# B&R Automation Studio project AS (part 2)

#### bgssm.c
```c
/********************************************************************
 * COPYRIGHT -- belgor
 ********************************************************************
 * Library: bglibas
 * File: bglibas.c
 * Author: admin
 * Created: March 07, 2012
 ********************************************************************
 * Implementation of library bglibas
 ********************************************************************/

#ifdef __cplusplus
  extern "C"
  {
#endif

#include <string.h>
// #include <stdarg.h>

#include  "bglibasWBR.h"                                                        //  WBR: could also keep the bglibas.h name and change the library's Properties->Library setting away from using the default name
#include  "bglibasWBR_C.h"

/* Init state machine. MUST be called once, before any other bgSSM function call. */
unsigned long bgSSMInit(struct bgSSM_typ* p, unsigned long pFunGetStateName, unsigned long pFunCyclicCallback)
{
  memset(p, 0, sizeof(struct bgSSM_typ));

  p->pfunGetStateName = (UDINT)pFunGetStateName;
  p->pfunCyclicCallback = (UDINT)pFunCyclicCallback;
  p->stateInit = 1;
  return(0);
}

/** Function pointer Init state machine. MUST be called once, before any other bgSSM function call. */
unsigned long bgSSMInitWbr(struct bgSSM_typ* p,                                    //  Pointer to state machine members and methods
                           unsigned long pfunInitState,                            //  Mandatory - initial method must be assigned
                           unsigned long pfunInterrupt,                            //  Optional
                           unsigned long pFunCyclicCallback)                       //  Optional
{
  memset(p, 0, sizeof(struct bgSSM_typ));

  p->pfunInitState=       (UDINT)pfunInitState;
  p->pfunInterrupt=       (UDINT)pfunInterrupt;
  p->pfunCyclicCallback=  (UDINT)pFunCyclicCallback;

  p->log.str.i.maxNodes=  200;
  p->log.str.list=  (linkedList_typ *)listSvcRequestList(BGSSM_MESSAGE_LENGTH_C,  lsQUEUE);

  p->stateNext= p->pfunInitState;                                                   //  WBR: assign init state function

  return(0);
}

/** State machine (SM) cyclic operation. */
unsigned long bgSSMCyclic(struct bgSSM_typ* p)
{
  int ii;

  //  TODO: implement interrupt/pause here to pause the delays with the SM

  //operate all timers
  for(ii=0; ii<BGSSM_TIMER_COUNT;ii++){
    bgTimerCyclic(&p->timer_x1ms[ii]);
  }
  bgTimerCyclic(&p->dlytimer_x1ms);
  bgTimerCyclic(&p->wdogTimer_x1ms);        //! \todo   log watchdog timeout \
                                                        provide automatic error state and go there? \
                                                        test func bgSSMStateNextWithWatchdog()

  //operate dlyCycle counter
  if(p->dlyCycles){
    p->dlyCycles--;
  }

  //call cyclic callback function if defined
  if(p->pfunCyclicCallback){
    void(*callback)(bgSSM_typ*) = ( void (*) (bgSSM_typ*) ) p->pfunCyclicCallback;
    (*callback)(p);
  }

  //clear single cycle flag every scan
  p->stateInit = 0;

  /// Evaluate breakpoint feature
  if(p->scanLimit.breakpoint && !p->scanLimit.active)   p->scanLimit.active=  1;          //  breakpoint has been found
  if(p->scanLimit.breakpointPrev && !p->scanLimit.breakpoint)   p->scanLimit.active=  0;  //  breakpoint switched off by

  /// Evaluate limit scan feature
  if(p->scanLimit.triggerNextScan)
  {
    p->scanLimit.triggerNextScan= p->scanLimit.count= 0;
  }
  if(!p->scanLimit.active)          memset(&p->scanLimit, 0, sizeof(p->scanLimit));
  else
  {
    if(p->scanLimit.count >= p->scanLimit.limit)   return 1;
    p->scanLimit.count++;
  }

  //check if state change requested
  if(p->state != p->stateNext){

    //if state change w. delay > wait for delay timer to expire or dlyCycles == 0
    if(!bgTimerIsTimeOut(&p->dlytimer_x1ms) || p->dlyCycles){                   //  TODO: add delay until event?
      return 1;
    }

    p->state = p->stateNext;
    //generate stateInit single scan flag
    p->stateInit = 1;

    //define state name if external function for state names is defined
    if( p->pfunGetStateName ){
      char*(*getStateName)(UDINT) = ( char* (*) (UDINT) )p->pfunGetStateName;
      strcpy(p->stateText, (*getStateName)(p->state));
    }else{
      strcpy(p->stateText, "???");
    }
  }

  if(p->pfunInitState)                                                          //  if the init state function pointer is defined...
  {
    void(*callState)(bgSSM_typ*) = ( void (*) (bgSSM_typ*) ) p->state;          //  ... call the function for the current state, i.e. use function pointer SM - WBR:
    (*callState)(p);
  }
  return(0);
}

/** SM state change methods
=============================*/

/** Change to next state. */
unsigned long bgSSMStateNext(struct bgSSM_typ* p, unsigned long stateNext)
{
  p->stateNext = stateNext;
  return(p->stateNext);
}

/** Store state to go to after SM subroutine. */
unsigned long bgSSMStateAfterSub(struct bgSSM_typ* p, unsigned long stateAfterSub)
{
  if(p->stateAfterSubIndex >= BGSSM_SUBROUTINE_COUNT)   return -99;     //  TODO: handle this error

  p->stateAfterSub[p->stateAfterSubIndex] = stateAfterSub;
  return(p->stateAfterSub[p->stateAfterSubIndex++]);
}

/** Activate state to go to after SM subroutine. */
unsigned long bgSSMReturnFromSub(struct bgSSM_typ* p)
{
  if(p->stateAfterSubIndex >= BGSSM_SUBROUTINE_COUNT)   return -99;     //  TODO: handle this error

  p->stateNext=    p->stateAfterSub[p->stateAfterSubIndex--];
  return(p->stateNext);
}

/** Change to next state w. timer delay. */
unsigned long bgSSMStateNextWithWatchdog(struct bgSSM_typ* p, unsigned long stateNext, unsigned long wdogTimeX1ms)
{
  p->stateNext = stateNext;
  bgTimerStart(&p->wdogTimer_x1ms, wdogTimeX1ms);
  return(p->stateNext);
}

/** Change to next state w. timer delay. */
unsigned long bgSSMStateNextTimeDelay(struct bgSSM_typ* p, unsigned long stateNext, unsigned long delayTimeX1ms)
{
  p->stateNext = stateNext;
  bgTimerStart(&p->dlytimer_x1ms, delayTimeX1ms);
  return(p->stateNext);
}

/** Change to next state w. cycles delay. */
unsigned long bgSSMStateNextCycleDelay(struct bgSSM_typ* p, unsigned long stateNext, unsigned long delayCycles)
{
  p->stateNext = stateNext;
  p->dlyCycles = delayCycles;
  return(p->stateNext);
}

/** Check if first scan for the state. */
plcbit bgSSMIsStateInit(struct bgSSM_typ* p)
{
  return(p->stateInit);
}

/** \todo  document */
UDINT  bgSSMPrintToTextLog(struct bgSSM_typ* p, const char* format, ...)
{
 va_list ap;

  va_start(ap, format);
  wbrvsnprintf((char *)listSvcRequestListNode(p->log.str.list), BGSSM_MESSAGE_LENGTH_C, format, ap);
  va_end(ap);

  return  listSvcCharListToStringArray(
                  p->log.str.list
                , &p->log.view[0][0]
                , BGSSM_MESSAGE_LENGTH_C
                , BGSSM_LOG_ENTRIES
                , p->log.str.i.offset
                , p->log.str.i.pageOffset
                , p->log.str.i.maxNodes
                , 1
                , ""
               );
}

/** \todo  document */
UDINT  bgSSMPrintLogMessage(struct bgSSM_typ* p)
{
  return  bgSSMPrintToTextLog(p, "%s", p->msg.log);
}

/** \todo  document */
UDINT  bgSSMPrintToTextLogIEC(struct bgSSM_typ* p, char* message)
{
  return  bgSSMPrintToTextLog(p, "%s", message);
}

/** \todo  document */
DINT  bgSSMPrintToLogbook(struct bgSSM_typ* p, const char* text, UDINT logIdent)
{
  return  requestMessageToLog( (UDINT)text, logIdent, 0, 0, 0, 0);              //  logIdent currently not used if logMsgType param is zero
}

/** \todo  document */
DINT  bgSSMPrintLogMessageToLogbook(struct bgSSM_typ* p, UDINT logIdent)    //! \todo   strcpy(loggermsg, requestedmsg) since msg gets destroyed, at least in ARsim
{
  return  requestMessageToLog( (UDINT)p->msg.log, logIdent, 0, 0, 0, 0);           //  logIdent currently not used if logMsgType param is zero
}

/** \todo  document */
DINT  bgSSMPrintToLogbookIEC(struct bgSSM_typ* p, char* message, UDINT logIdent)    //! \todo   strcpy(loggermsg, requestedmsg) since msg gets destroyed, at least in ARsim
{
  return  requestMessageToLog( (UDINT)message, logIdent, 0, 0, 0, 0);           //  logIdent currently not used if logMsgType param is zero
}

/** Check if first scan for the state.  If yes, perform some standard state change functions */
BOOL bgSSMIsStateInitWBR( struct bgSSM_typ* p                    //!  \todo   move this to C header
                        , /* const */ char* stateText            //!< This can take __FUNCTION__ or "text"
                        )
{
  if(p->stateInit)
  {
    if(stateText)  strcpy(p->stateText, stateText);
    wbrsnprintf(p->msg.log, sizeof(p->msg.log), "%s(%d)", bgSSMGetStateText(p), bgSSMGetState(p));      //! \todone? reserve p->message for other messages?
    bgSSMPrintToTextLog(p, "%s", p->msg.log);
    bgSSMPrintToLogbook(p, p->msg.log, 1);
  }

  return(p->stateInit);
}

/** SM data retrieval methods
=============================*/

/** Get current state */
unsigned long bgSSMGetState(struct bgSSM_typ* p)
{
  return(p->state);
}

/** Get current state text*/
plcstring* bgSSMGetStateText(struct bgSSM_typ* p)
{
  return(&p->stateText[0]);
}

#ifdef __cplusplus
  };
#endif
```

### Library Logical/UserLibraries/wbrServices/wbrPingSvc (ANSIC) - Ping a host or IP address
Depends on: AsICMP, wbrLogSvc, bglibasWBR, AsTime

### Package Logical/UserLibraries/wbrServices/wbrSvcUtilities - Utility functions

- Library Logical/UserLibraries/wbrServices/wbrSvcUtilities/wbrBitUtil (ANSIC) - Utilities for setting or extracting bits in bytes, words, ints, etc. (no source held here)

### wbrServicesGlobal.var - Global variables
```iecst
(********************************************************************
 * COPYRIGHT -- Piedmont Automation
 ********************************************************************
 * Package: listServices
 * File: listServicesGlobal.var
 * Author: Blanton Radford
 * Created: August 11, 2014
 ********************************************************************
 * Variables of package listServices
 ********************************************************************)
VAR
	memService : wbrMemService_typ := (0);
	logService : wbrLogService_typ := (0);
	genericPing : wbrPingService_typ;
	usbServiceIF : ARRAY[0..wbrusbLAST_NODE] OF wbrUSBServiceIF_typ;
END_VAR
```

### wbrServicesPackage.var - Package variables
```iecst
VAR
	usbService : wbrUSBService_typ;
END_VAR
```

### Package Logical/UserLibraries/wbrServices/InitSP - Place this program in TC#1 to initialize wbrServices

### paiConfig.typ
```iecst
(********************************************************************
 * COPYRIGHT --
 ********************************************************************
 * Package: ConfigAndRecipes
 * File: Config.typ
 * Author: goran_2
 * Created: August 06, 2011
 ********************************************************************
 * Data types of package ConfigAndRecipes
 ********************************************************************)
(*==================================================================*)
(*Config related structures that shall not be changed.*)
(*==================================================================*)

TYPE
	cfgConfig_enums :
		(
		ENUM_APPCFG_INFO_TEXT_LEN := 127,
		ENUM_APPCFG_PATHNAME_MAXLEN := 64,
		ENUM_APPCFG_PWD_MAXLEN := 15,
		ENUM_APPCFG_DEFECT_MAXINDEX := 11,
		ENUM_APPCFG_DEFECT_TXTMAXLEN := 31,
		ENUM_APPCFG_MAGIC_NUMBER := 16#55555555 (*Magic word (010101...) sequence (to detect battery backed up memory alterations)*)
		);
	cfgConfig_typ : 	STRUCT  (*Machine configuration includes settings for timers and settings for servo drives.*)
		cfgDefault : cfgMachineConfig_typ; (*The hardcoded defaults from the various application tasks.  This config should not be written to in the application code.  \todo  maintain a separate config that is the factory default config?*)
		machine : cfgMachineConfig_typ; (*The machine-level config.  Any item not set as product-level will use the value from this config.  When a different product is activated, this config will be copied to the active config first.*)
		recipe : cfgMachineConfig_typ; (*A holding space for a non-active recipe, i.e. product, config.  Possibly not needed or better located in the HMI package.  Would be used to support HMI editing of a product config that is not the active config.*)
		active : cfgMachineConfig_typ; (*The config used for current machine operation.  This will be the machine config*)
	END_STRUCT;
END_TYPE
```

### ConfigAndRecipes.var
```iecst
(********************************************************************
 * COPYRIGHT --
 ********************************************************************
 * Package: ConfigAndRecipes
 * File: ConfigAndRecipes.var
 * Author: goran_2
 * Created: August 06, 2011
 ********************************************************************
 * Variables of package ConfigAndRecipes
 ********************************************************************)
(*Constants*)
VAR CONSTANT
	APPCFG_DIRPATH_MAXLEN_IEC : DINT := 47;
	APPCFG_DIRPATH_MAXLEN_C : DINT := APPCFG_DIRPATH_MAXLEN_IEC + 1;
	APPCFG_FILENAME_MAXLEN_IEC : DINT := 63;
	APPCFG_FILENAME_MAXLEN_C : DINT := APPCFG_FILENAME_MAXLEN_IEC + 1;
	APPCFG_EXTENSION_MAXLEN_IEC : DINT := 15;
	APPCFG_EXTENSION_MAXLEN_C : DINT := APPCFG_EXTENSION_MAXLEN_IEC + 1;
	APPCFG_FULLPATH_MAXLEN_C : DINT := APPCFG_DIRPATH_MAXLEN_C + APPCFG_FILENAME_MAXLEN_C + APPCFG_EXTENSION_MAXLEN_C;
	APPCFG_FULLPATH_MAXLEN_IEC : DINT := APPCFG_FULLPATH_MAXLEN_C - 1;
END_VAR
(*Variables*)
VAR
	gConfig : cfgConfig_typ := (0); (*Machine configuration data*)
END_VAR
```

### Program Logical/UserLibraries/wbrServices/InitSP/runFirst (ANSIC) - Init wbrServices - PLACE IN TC#1 above most if not all other tasks

#### runFirstInit.c
```c
/*!
 ********************************************************************
 * Program : runFirst
 * \file :   runFirstInit.c
 * \author : Blanton Radford
 * \date Created: May 07, 2015
 * \copyright -- Piedmont Automation
 ********************************************************************
 * \brief Initializations for package WBRServices
 ********************************************************************/

#ifdef _DEFAULT_INCLUDES
  #include <AsDefault.h>
#endif

/*! \brief Init project compile info
*   called only from runFirstInit
*/
static void wbrServiceInitProgramCompileInfo()
{
 char osVers[12];
 TARGETInfo_typ TInfo;

  TInfo.enable = 1;
  TInfo.pOSVersion = (UDINT) &osVers;

  do {
    TARGETInfo(&TInfo);
  } while(TInfo.status == 0xFFFF);

#ifndef AS_PROJ
  #warning Macro names for program complile info not defined \
           -- code located just below this warning
  wbrsnprintf(gConfig.cfgDefault.cfgCompile.info, sizeof(gConfig.cfgDefault.cfgCompile.info), "No compile info");
  //* Copy the line below into Project->Change Runtime Versions->Build->ANSI C Build Options to define \
         -D "str(x)=#x" -D AS_PROJ=str($(AS_PROJECT_NAME)) -D AS_CFG=str($(AS_CONFIGURATION)) -D "AS_VERS=str($(AS_VERSION))" -D "AS_USER=str($(AS_USER_NAME))" -D "AS_CMPNY=str($(AS_COMPANY_NAME))" -D "AS_BUILD_MODE=str($(AS_BUILD_MODE))"

#else
  // These macro names are defined in Project->Change Runtime Versions->
  //    Build->ANSI C Build Options
  wbrsnprintf(gConfig.cfgDefault.cfgCompile.projVersion,  sizeof(gConfig.cfgDefault.cfgCompile.projVersion),  "%s, V1.0.00.6",  AS_PROJ);
  wbrsnprintf(gConfig.cfgDefault.cfgCompile.AS_config,    sizeof(gConfig.cfgDefault.cfgCompile.AS_config),    "%s",             AS_CFG);
  wbrsnprintf(gConfig.cfgDefault.cfgCompile.AS_configID,  sizeof(gConfig.cfgDefault.cfgCompile.AS_configID),  "%s_%s",          AS_PROJ, AS_CFG);
  wbrsnprintf(gConfig.cfgDefault.cfgCompile.AS_build,     sizeof(gConfig.cfgDefault.cfgCompile.AS_build),     "%s",             AS_BUILD_MODE);
  wbrsnprintf(gConfig.cfgDefault.cfgCompile.date,         sizeof(gConfig.cfgDefault.cfgCompile.date),         "%s @ %s",        __DATE__, __TIME__);
  wbrsnprintf(gConfig.cfgDefault.cfgCompile.AS_version,   sizeof(gConfig.cfgDefault.cfgCompile.AS_version),   "%s",             AS_VERS);
  wbrsnprintf(gConfig.cfgDefault.cfgCompile.user,         sizeof(gConfig.cfgDefault.cfgCompile.user),         "%s",             AS_USER);
  wbrsnprintf(gConfig.cfgDefault.cfgCompile.company,      sizeof(gConfig.cfgDefault.cfgCompile.company),      "%s, Inc.",       AS_CMPNY);
  wbrsnprintf(gConfig.cfgDefault.cfgCompile.info,         sizeof(gConfig.cfgDefault.cfgCompile.info),         "Compile info complete");
#endif
  wbrsnprintf(gConfig.cfgDefault.cfgCompile.AR_Version,   sizeof(gConfig.cfgDefault.cfgCompile.AR_Version),   "%s",           osVers);
  //! \todo   add WBRServices version, drawing name and revision, SVN revision
}

/*! \brief Init machine configuration defaults
*   called only from runFirstInit
*/
void  wbrMemServiceFirstInitSetDefaults(wbrMemSvcStoredConfig_typ* cfg)
{
  cfg->memRequestSize=   0xFFFFFF;

//  if(gREMMEMPostfix == 0x55555555)                                                 //  if storage has data, ...
//    cfg->memRequestSize=  (gRemanentData.activeCfg.wbrMemService.memRequestSize > 0xFFFFFF) ? gRemanentData.activeCfg.wbrMemService.memRequestSize : 0xFFFFFF;
  // if(magic == 0x55555555)                          //  if storage has data, ...
    // cfg->memRequestSize=  stored.wbrMemService.memRequestSize;
}

/*! \brief Init-SP for AsMem heap memory and linked list services
*   \pre   Place in TC#1 in front of most if not all other tasks
*/
void _INIT runFirstInit(void)
{
  wbrServiceInitProgramCompileInfo();

  //! \todo init AsMem as a separate service
  //! \todo what to do with appConfigAndRec - switch to MAPP?

  /// Init cfgDefault with hardcoded defaults
  if(&gConfig.cfgDefault.wbrMemService != 0)                   //  mcfgWBR: skip if this address is null    TODO: log this for debug
    memService.config= &gConfig.cfgDefault.wbrMemService;                //  mcfgWBR: this needs to run before the Config & Recipe task to insure the defaults are set

    // memService.config= &config.wbrMemService;                               //  mcfgWBR: used only for testing package independently

  wbrMemServiceFirstInitSetDefaults(memService.config);

  memService.status.memInitValid= initMemSvc(memService.config->memRequestSize);

  initListSvc(memService.status.memInitValid);

  setLogServiceDataAddress(&logService);

  if(memService.status.memInitValid)       initLogService();

  requestMessageToLogDefault( (UDINT)gConfig.cfgDefault.cfgCompile.projVersion);
  requestMessageToLogDefault( (UDINT)gConfig.cfgDefault.cfgCompile.AS_config);
  requestMessageToLogDefault( (UDINT)gConfig.cfgDefault.cfgCompile.AS_configID);
  requestMessageToLogDefault( (UDINT)gConfig.cfgDefault.cfgCompile.AS_build);
  requestMessageToLogDefault( (UDINT)gConfig.cfgDefault.cfgCompile.date);
  requestMessageToLogDefault( (UDINT)gConfig.cfgDefault.cfgCompile.AS_version);
  requestMessageToLogDefault( (UDINT)gConfig.cfgDefault.cfgCompile.AR_Version);
  requestMessageToLogDefault( (UDINT)gConfig.cfgDefault.cfgCompile.user);
  requestMessageToLogDefault( (UDINT)gConfig.cfgDefault.cfgCompile.company);
  requestMessageToLogDefault( (UDINT)gConfig.cfgDefault.cfgCompile.info);
  requestMessageToLogDefault( (UDINT)"wbrServices v0.12.0 initialized");
  requestSuccessEventToLog(
                        (UDINT)__FUNCTION__
                      , getSystemUserLogIdent()
                      , 0
                      , 50000
                      , 0
                      , (UDINT)"wbrServices v0.12.0 initialized"
                      , sizeof("wbrServices vn.nn.n initialized")
                      );

  wbrPingSvcInit(&genericPing);
}
```


### Package Logical/UserLibraries/wbrServices/TimerServices - ms-based time counters, pulses, etc.

### TimerServices.typ
```iecst
(********************************************************************
 * COPYRIGHT -- Piedmont Automation
 ********************************************************************
 * Package: TimerServices
 * File: TimerServices.typ
 * Author: Blanton Radford
 * Created: December 05, 2014
 ********************************************************************
 * Data types of package TimerServices
 ********************************************************************)

TYPE
	mstpPERIOD_enum :
		(
		per00100 := 0,
		per00200,
		per00500,
		per01000,
		per02000,
		per05000,
		per10000,
		perLAST
		);
	mstpFREQUENCY_enum :
		(
		freq010Hz := 0,
		freq005Hz,
		freq002Hz,
		freq001Hz,
		freq0p5Hz,
		freq0p2Hz,
		freq0p1Hz,
		freqLAST
		);
	mstpDUTY_CYCLE_enum :
		(
		duty01 := 0,
		duty10,
		duty20,
		duty25,
		duty50,
		dutyLAST
		);
	mstpDURATION_enum :
		(
		dur001ms := 0,
		dur010ms,
		dur020ms,
		durLAST
		);
	msTimerHourMeter_typ : 	STRUCT
		enable : BOOL;
		count : UDINT;
	END_STRUCT;
	msTmPulseSOS_typ : 	STRUCT
		codeSignal : BOOL;
		msgEnable : BOOL;
		shortEnable : BOOL;
		longEnable : BOOL;
		shortPulse : BOOL;
		longPulse : BOOL;
	END_STRUCT;
	msTmPulsePeriodDutyInOut_typ : 	STRUCT
		iPeriodValue : UDINT;
		iDutyValue : REAL;
		oPulse : BOOL;
	END_STRUCT;
	msTmPulseFreqDutyInOut_typ : 	STRUCT
		iFreqValue : REAL;
		iDutyValue : REAL;
		oPulse : BOOL;
	END_STRUCT;
	mstpPerDutyDurTableElements_typ : 	STRUCT
		duty : {REDUND_UNREPLICABLE} ARRAY[0..dutyLAST]OF BOOL;
		duration : {REDUND_UNREPLICABLE} ARRAY[0..durLAST]OF BOOL;
	END_STRUCT;
	msTimerPulse_typ : 	STRUCT
		periodDutyDurationTable : {REDUND_UNREPLICABLE} ARRAY[0..perLAST]OF mstpPerDutyDurTableElements_typ;
		periodLength : USINT;
		sos : msTmPulseSOS_typ;
	END_STRUCT;
	msTimer_typ : 	STRUCT
		pulse : msTimerPulse_typ; (*Various pulses calculated with ms precision (when allowed to by task class timing)*)
		initVal : UDINT; (*Initial value of clock_ms*)
		rolloverVal : UDINT;
		clock_ms : UDINT; (*System ms counter.  Not resettable.  Used to keep C1ms from missing counts if task class runs into its tolerance  TODO:  \todo*)
		diff_ms : UDINT; (*Difference from one scan to the next of the msTimeSvc task*)
		C1ms : UDINT; (*Rolls over after 4294920000U to keep other Cxx counters accurate.  Can also be reset.*)
		C10ms : UDINT;
		C100ms : UDINT;
		C1s : UDINT;
		C10s : UDINT;
		C60s : UDINT;
		C01sAbs : UDINT;
		C60sAbs : UDINT;
		F100ms : BOOL;
		F500ms : BOOL;
		F1s : BOOL;
		F2s : BOOL;
		F10s : BOOL;
		pulse01Hz100ms : BOOL;
		pulse1day100ms : BOOL;
		prev60s : UDINT;
		prev01s : UDINT;
	END_STRUCT;
END_TYPE
```

### Program Logical/UserLibraries/wbrServices/TimerServices/msTimeSvc (ANSIC)

#### msTimeSvc.c - Implementation code
```c
/*!
 ********************************************************************
### Program : msTimeSvc
 * \file :   msTimeSvc.c
 * \author : Blanton Radford
 * \date Created: December 05, 2014
 * \copyright -- Piedmont Automation
 ********************************************************************
 * \brief Implementation of program msTimeSvc
 ********************************************************************/

#ifdef _DEFAULT_INCLUDES
  #include <AsDefault.h>
#endif

_LOCAL BOOL running;    //  temporary
_LOCAL UDINT  run_ms;   //  temp

msTimer_typ * t=  &msTimer;

msTmPulsePeriodDutyInOut_typ  periodDutyDurationTable[perLAST][dutyLAST + durLAST]=
{
  {
      {  100,  1.0, 0}        //  period in ms, duty cycle in Hz, output
    , {  100, 10.0, 0}
    , {  100, 20.0, 0}
    , {  100, 25.0, 0}
    , {  100, 50.0, 0}
    , {  100, 01.0, 0}        //  period in ms, duty cycle in Hz, output
    , {  100, 10.0, 0}
    , {  100, 20.0, 0}
  }
 ,{
      {  200,  1.0, 0}        //  period, duty cycle, output
    , {  200, 10.0, 0}
    , {  200, 20.0, 0}
    , {  200, 25.0, 0}
    , {  200, 50.0, 0}
    , {  200, 01.0, 0}        //  period, duration, output
    , {  200, 10.0, 0}
    , {  200, 20.0, 0}
  }
 ,{
      {  500,  1.0, 0}        //  period, duty cycle, output
    , {  500, 10.0, 0}
    , {  500, 20.0, 0}
    , {  500, 25.0, 0}
    , {  500, 50.0, 0}
    , {  500, 01.0, 0}        //  period, duration, output
    , {  500, 10.0, 0}
    , {  500, 20.0, 0}
  }
 ,{
      { 1000,  1.0, 0}        //  period, duty cycle, output
    , { 1000, 10.0, 0}
    , { 1000, 20.0, 0}
    , { 1000, 25.0, 0}
    , { 1000, 50.0, 0}
    , { 1000, 01.0, 0}        //  period, duration, output
    , { 1000, 10.0, 0}
    , { 1000, 20.0, 0}
  }
 ,{
      { 2000,  1.0, 0}        //  period, duty cycle, output
    , { 2000, 10.0, 0}
    , { 2000, 20.0, 0}
    , { 2000, 25.0, 0}
    , { 2000, 50.0, 0}
    , { 2000, 01.0, 0}        //  period, duration, output
    , { 2000, 10.0, 0}
    , { 2000, 20.0, 0}
  }
 ,{
      { 5000,  1.0, 0}        //  period, duty cycle, output
    , { 5000, 10.0, 0}
    , { 5000, 20.0, 0}
    , { 5000, 25.0, 0}
    , { 5000, 50.0, 0}
    , { 5000, 01.0, 0}        //  period, duration, output
    , { 5000, 10.0, 0}
    , { 5000, 20.0, 0}
  }
 ,{
      {10000,  1.0, 0}        //  period, duty cycle, output
    , {10000, 10.0, 0}
    , {10000, 20.0, 0}
    , {10000, 25.0, 0}
    , {10000, 50.0, 0}
    , {10000, 01.0, 0}        //  period, duration, output
    , {10000, 10.0, 0}
    , {10000, 20.0, 0}
  }
}  ;

static  BOOL  pulsePeriodDurationWithOffset(
          UDINT per     //  period in ms
        , UDINT dur     //  Duration ( pulse on time) in ms
        , UDINT off     //  offset of start of pulse in ms
        )
{
  if(per < 2)   return  0;                                                      //  Period must be at least 2ms using ms precision
                                                                                //  Period must also be at least 2 * TC cycle time
  return  (   ((t->C1ms % per) >= off)
           && ((t->C1ms % per) < dur + off));
}

BOOL  getPulseOfPeriodAndDurationWithOffset(
          UDINT per     //  period in ms
        , UDINT dur     //  Duration ( pulse on time) in ms
        , UDINT off     //  offset of start of pulse in ms
        )
{
  return  pulsePeriodDurationWithOffset(per, dur, off);
}

BOOL  pulsePeriodDuration(
          UDINT per     //  period in ms
        , UDINT dur     //  Duration ( pulse on time) in ms
        )
{
  return  pulsePeriodDurationWithOffset(per, dur, 0);
}

BOOL  pulsePeriodDuty(
          UDINT per     //  period in ms
        , REAL  duty    //  duty cycle in %
        )
{
  if(duty <= 0.0)      return  0;                                                  //  Duty cycle must be greater than zero
  if(duty >= 100.0)    return  1;                                                  //  Signal always on if duty greater than 100%

  return  pulsePeriodDurationWithOffset(
                        per
                      , (UDINT)((REAL)per * duty / 100.0)
                      , 0
                      );
}

BOOL  pulseFreqDuty(
          REAL  f       //  frequency in Hz
        , REAL  d       //  duty cycle in %
        )
{
  if(d <= 0.0)      return  0;                                                  //  Duty cycle must be greater than zero
  if(f <= 0.0)      return  0;                                                  //  Prevent divide by zero
  if(f > 500.0)     return  0;                                                  //  Can't process higher frequencies using ms precision

  if(d >= 100.0)    return  1;                                                  //  Signal always on if duty greater than 100%

  return  pulsePeriodDurationWithOffset(
                        (UDINT)(1000.0 / f)
                      , ((UDINT)(1000.0 / f) * d / 100.0)
                      , 0
                      );
}

BOOL  pulseFreqDutyWithOffset(
          REAL  f       //  frequency in Hz
        , REAL  d       //  duty cycle in %
        , REAL  o       //  offset of start of pulse in %
        )
{
  if(d <= 0.0)      return  0;                                                  //  Duty cycle must be greater than zero
  if(f <= 0.0)      return  0;                                                  //  Prevent divide by zero
  if(f > 500.0)     return  0;                                                  //  Can't process higher frequencies using ms precision

  if(d >= 100.0)                  return  1;                                    //  Signal always on if duty greater than 100%
  if(o >= 100.0)                  return  0;                                    //  Signal always off if offset greater than 100%

  return  pulsePeriodDurationWithOffset(
                        (UDINT)(1000.0 / f)
                      , ((UDINT)(1000.0 / f) * d / 100.0)
                      , ((UDINT)(1000.0 / f) * o / 100.0)
                      );
}

BOOL  pulseFreqDuration(
          REAL  f       //  frequency in Hz
        , UDINT dur     //  Duration ( pulse on time) in ms
        )
{
  if((f <= 0.0) || (f > 500.0))   return  0;

  return  pulsePeriodDurationWithOffset(
                        (UDINT)(1000.0 / f)
                      , dur
                      , 0
                      );
}

BOOL  pulseFreqDurationWithOffset(
          REAL  f       //  frequency in Hz
        , UDINT dur     //  Duration ( pulse on time) in ms
        , UDINT off     //  offset of start of pulse in ms
        )
{
  if((f <= 0.0) || (f > 333.33))   return  0;

  return  pulsePeriodDurationWithOffset(
                        (UDINT)(1000.0 / f)
                      , dur
                      , off
                      );
}

/*! \brief Init-SP for millisecond timer services
*   \pre   Place in TC#1 or first used TC
*/
void _INIT msTimeSvcInit(void)
{

}

/*! \brief Cyclic task for millisecond timer services
*   \pre   Place in TC#1 or first used TC
*/
void _CYCLIC msTimeSvcCyclic(void)
{
 int  i, j;

  if(t->clock_ms == 0)    t->initVal= (UDINT)clock_ms();

  // if(<use external clock>)
  // t->clock_external=  <count from external source>;  i.e. a TC of < 1ms duration

  t->clock_ms=  (UDINT)clock_ms();

  t->diff_ms= t->clock_ms - t->C1ms - t->initVal;   //  Will this work at rollover?

  t->C1ms=  t->clock_ms - t->initVal; // + <rolloverVal>

  //! \todo   update C1ms in case task class runs into its tolerance \
              do this using a diff calc so that the function will continue to operate even if C1ms rolls over \
              OR just use clock_ms time and live with the rollover or implement a rollover counter

  /*! \todo
      if(<rolloverActive>)
        <rolloverVal>=  t->clock_ms - t->initVal + <prevRolloverVal> - 4294920000U;

      if( !<rolloverActive> && (t->C1ms > 4294920000U))
        <prevRolloverVal>=  <rolloverVal>;
        <rolloverVal>=  t->C1ms - 4294920000U;
        XX t->C1ms=  t->clock_ms=  0;      //  Keep absolute minute count accurate - WBR: check to see if this works
        XX -- OR --
        t->C1ms=  <rolloverVal>;      //  Keep absolute minute count accurate - WBR: check to see if this works
        t->C01sAbs++;
        t->C60sAbs++;
        rolloverActive= 1;

      //  This code will likely need to move ahead of t->diff_ms assignment
      if(t->clock_ms < t->C1ms)     //  rolled over
        t->initVal= (UDINT)clock_ms();
        <rolloverVal>+= t->diff_ms;  // assuming diff_ms works at rollover
        rolloverActive= 0;
        assign t->C1ms as above
  */
  // t->C1ms++;                                // inc ms counter
                                            // this will roll over after
                                            // 49.7102 days of continuous
                                            // running - WBR
                                            // resets with Start button

  /// Calculate Other Counters
  t->C10ms=   t->C1ms /   10;
  t->C100ms=  t->C1ms /  100;
  t->C1s=     t->C1ms / 1000;
  t->C10s=    t->C1ms / 10000;
  t->C60s=    t->C1ms / 60000;

  if(t->C1s  > t->prev01s)    t->C01sAbs++;       //  Rolls over after 136.193 years
  if(t->C60s > t->prev60s)    t->C60sAbs++;       //  Rolls over after 8171.55 years

  t->prev01s=  t->C1s;
  t->prev60s=  t->C60s;

  ///  Calc pulse trains
  //  <boolean>=    ((t->C1ms % <period>) < <duration>);      //  example - period and duration are in ms

  for(i=0; i<perLAST; i++)
  {
    for(j=0; j<dutyLAST; j++)
    {
      t->pulse.periodDutyDurationTable[i].duty[j]=
      periodDutyDurationTable[i][j].oPulse=
        pulsePeriodDuty(
            periodDutyDurationTable[i][j].iPeriodValue
          , periodDutyDurationTable[i][j].iDutyValue
          );
    }
    for( ; j < durLAST + dutyLAST; j++)
    {
      t->pulse.periodDutyDurationTable[i].duration[j - dutyLAST]=
      periodDutyDurationTable[i][j].oPulse=
        pulsePeriodDuration(
            periodDutyDurationTable[i][j].iPeriodValue
          , periodDutyDurationTable[i][j].iDutyValue
          );
    }
  }

  //  new
  t->pulse01Hz100ms= pulsePeriodDuration(1000, 100);                              //  add these in the application as needed, or put frequently used ones here
  t->pulse1day100ms= pulsePeriodDuration((24*3600*1000), 100);                    //  comes on once per day for 100ms

  t->pulse.sos.msgEnable=   pulseFreqDuty(0.25, 75.0);
  t->pulse.sos.shortEnable= pulseFreqDuty(0.50,  35.0);
  t->pulse.sos.longEnable=  pulseFreqDutyWithOffset(0.25, 17.5, 25.0);
  t->pulse.sos.shortPulse=  pulseFreqDuty( 4.0,  20.0);
  t->pulse.sos.longPulse=   pulseFreqDuty( 4.0,  60.0);

  t->pulse.sos.codeSignal=
    (   (t->pulse.sos.msgEnable && t->pulse.sos.shortEnable && t->pulse.sos.shortPulse)
     || (t->pulse.sos.msgEnable && t->pulse.sos.longEnable && t->pulse.sos.longPulse)) ;

  //  legacy
  t->F100ms=  pulsePeriodDurationWithOffset(  100,   50, 0);
  t->F500ms=  pulsePeriodDurationWithOffset(  500,  250, 0);
  t->F1s=     pulsePeriodDurationWithOffset( 1000,  500, 0);
  t->F2s=     pulsePeriodDurationWithOffset( 2000, 1000, 0);
  t->F10s=    pulsePeriodDurationWithOffset(10000, 5000, 0);

  //  TODO: add configurable, periodic pulse(s), i.e. an (n)s pulse every (nn)min or (nn)day(s) or ???
  //  TODO: add hour meter(s)
  if(running)
  {
    run_ms+=  t->diff_ms;
  }
}
```

### varPkg.var
```iecst
VAR
	gMachine : HERNON_Inline_Machine_typ;
	gMachineType : HERNON_Machine_Types_Enum;
END_VAR
```

### Disp_Global_Var.var
```iecst
VAR
	gHMITable_Rec_Dispense : hmiTableFBK_typ;
	gHMITable_Cfg_Dispense : hmiTableFBK_typ;
END_VAR
```

- Program Logical/Application_Logic/pkgDispense/Dispense (IEC) - Manage all dispense-valve related functionality (IO slice DS1) (no source held here)

### Library Logical/Application_Logic/pkgDispense/libDisp (IEC)

#### Disp_Rec_Cfg.typ
```iecst
TYPE
	HERNON_Rec_Dispense_typ : 	STRUCT
		Enable : UDINT;
		Disp_Valve_Edgemode_Pulse_TO_ms : REAL;
		Enable_Cure : UDINT;
		Extra_Shots_Per_VBlock : UDINT;
		Vblock_Offset_Additional_Shots : ARRAY[0..MAX_IDX_MULTIPLE_DISPENSE_SHOTS]OF REAL;
	END_STRUCT;
	HERNON_Cfg_Dispense_typ : 	STRUCT
		VBlock_Offset_From_PiP_Sensor : UDINT;
		Disp_Valve_Max_Output_High_TO_S : REAL;
		Disp_Signal_Reset_MaxTO_S : REAL;
		Disp_Valve_Max_RDY_NegEdge_S : REAL;
		Disp_Output_NegEdge_Margin_S : REAL;
	END_STRUCT;
END_TYPE
```

#### Disp_IO.typ
```iecst
TYPE
	X20DS4389_Edgegen_typ : 	STRUCT
		iEdgeMasterTime : DINT;
		iReadOutputStatus : BOOL;
		oEnableEdgeGen : BOOL;
		iEdgeGenReadbackEnabled : BOOL;
		oEdgeGenSequence : SINT;
		iEdgegenSequenceReadback : SINT;
		oEdgeGenTimestamp : DINT;
		iEdgeGenError : BOOL;
		oQuitEdgeGenError : BOOL;
		iEdgeGenWarning : BOOL;
		oQuitEdgeGenWarning : BOOL;
	END_STRUCT;
	HERNON_Inline_Dispense_Item_typ : 	STRUCT
		iValveReady : BOOL;
		oDispTrigger : BOOL;
		EdgeGen : X20DS4389_Edgegen_typ;
	END_STRUCT;
	HERNON_Inline_Dispense_IO_typ : 	STRUCT
		Projectile : HERNON_Inline_Dispense_Item_typ;
		Primer : HERNON_Inline_Dispense_Item_typ;
		iEdgeDetectError : BOOL;
		oQuitEdgeDetectError : BOOL;
	END_STRUCT;
END_TYPE
```

#### Disp_Alarms_Warnings.typ
```iecst
TYPE
	HERNON_Alarm_Dispense_typ : 	STRUCT
		Valve_Error_1 : BOOL; (*0*)
		Valve_Not_On : BOOL; (*1*)
		Valve_Not_OFF : BOOL; (*2*)
		Dispense_Reset_Error : BOOL; (*3*)
		Valve_Not_Off : BOOL; (*4*)
		Err_Disp_VBlock_Acc_Idx : BOOL; (*5*)
		Dispense_IO_Alloc_Error : BOOL; (*6*)
		Disp_Output_Not_Reset : BOOL; (*7*)
		Dispense_ValveRdy_NegEdge_Err : BOOL; (*8*)
		Disp_Valve_On_Too_Long : BOOL; (*9*)
		Dispense_Twice_Single_VBlock : BOOL; (*10*)
		ValveRdy_Not_Reset : BOOL; (*11*)
		Dispense_Not_Ready_On_Start : BOOL; (*12*)
		Dispense_Error_During_Runtime : BOOL; (*13*)
		VBlock_idx_during_shot_wait : BOOL; (*14*)
		VBlock_Offset_Invalid : BOOL; (*15*)
	END_STRUCT;
END_TYPE
```

### Insp_Global_Var.var
```iecst
VAR
	gHMITable_Rec_Inspect : hmiTableFBK_typ;
	gHMITable_Cfg_Inspect : hmiTableFBK_typ;
END_VAR
```

### Program Logical/Application_Logic/pkgInspect/Inspect (IEC)

#### Main.st - Init, cyclic, exit code
```iecst
//     __ __                         __  ___               ___         __           _             ____
//    / // /__ _______  ___  ___    /  |/  /__ ____  __ __/ _/__ _____/ /___ ______(_)__  ___ _  /  _/__  ____
//   / _  / -_) __/ _ \/ _ \/ _ \  / /|_/ / _ `/ _ \/ // / _/ _ `/ __/ __/ // / __/ / _ \/ _ `/ _/ // _ \/ __/
//  /_//_/\__/_/ /_//_/\___/_//_/ /_/  /_/\_,_/_//_/\_,_/_/ \_,_/\__/\__/\_,_/_/ /_/_//_/\_, / /___/_//_/\__(_)
//                                                                                      /___/
//  Copyright

PROGRAM _INIT
	Init_Logbook.Enable := TRUE;
	Init_Logbook.Name := 'usr_insp';
	Init_Logbook();

	gHMITable_Rec_Inspect(tableName := 'REC_INSPECT',		nameSpace := 'hmiTable/Rec/Inspect',	Logbook := Init_Logbook.pLog, 		pOverallStats := ADR(gTableStats.Overall));
	gHMITable_Cfg_Inspect(tableName := 'CFG_INSPECT',		nameSpace := 'hmiTable/Cfg/Inspect',	Logbook := Init_Logbook.pLog, 		pOverallStats := ADR(gTableStats.Overall));
END_PROGRAM

PROGRAM _CYCLIC

END_PROGRAM

PROGRAM _EXIT

END_PROGRAM
```

#### Variables.var - Local variables
```iecst
VAR
	FBK_Inspection_Camera : ARRAY[0..MAX_IDX_INSPECT_UNITS] OF Hernon_Inspection_Camera;
	Init_Logbook : FBK_Init_Logbook;
END_VAR
```

#### LocalFunctions.fun
```iecst
FUNCTION_BLOCK Hernon_Inspection_Camera (*TODO: Add your comment here*) (*$GROUP=User,$CAT=User,$GROUPICON=User.png,$CATICON=User.png*)
	VAR_INPUT
		pInspectionIO : REFERENCE TO HERNON_Inline_Inspect_Item_typ;
		pInspVBlock : REFERENCE TO VBlock_Object_typ;
		pInspRec : REFERENCE TO HERNON_Rec_Inspect_typ;
		pInspCfg : REFERENCE TO HERNON_Cfg_Inspect_typ;
		pInspStats : REFERENCE TO HERNON_Prcs_Stats_typ;
		pMechanics : REFERENCE TO HERNON_Cfg_Mechanics_typ;
		pInspSeqFails : REFERENCE TO UDINT;
		MachineState : Global_State_Enum;
		VBlock_Fractional_Position : REAL;
		Current_VBlock_At_PiP_Sensor : UDINT;
		idx_inspect_unit : USINT;
	END_VAR
	VAR
		InspVar_LastCycle : HERNON_Inspect_App_typ;
		InspVar : HERNON_Inspect_App_typ;
		Alarms : HERNON_Alarm_Inspect_typ;
	END_VAR
END_FUNCTION_BLOCK
```

#### FBK_Inspection_Camera.st
```iecst
(* TODO: Add your comment here *)
FUNCTION_BLOCK Hernon_Inspection_Camera

	InspVar.VBlock_At_Inspect_Unit := (Current_VBlock_At_PiP_Sensor + (pMechanics.N_VBlocks_Belt_Total - pInspCfg.VBlock_Offset_From_PiP_Sensor)) MOD (pMechanics.N_VBlocks_Belt_Total);
	InspVar.VBlock_Fract_Pos := VBlock_Fractional_Position;

	CASE InspVar.Status OF
		INSPECT_STATE_INIT:
			pInspectionIO.oInspectionTrigger := FALSE;
			pInspectionIO.oIlluminationTrigger := FALSE;

			InspVar.Status := INSPECT_STATE_READY;

		INSPECT_STATE_READY:
			IF pInspRec.Enable = 1 THEN //If inspection is enabled:
				IF (InspVar.VBlock_At_Inspect_Unit <> InspVar_LastCycle.VBlock_At_Inspect_Unit) THEN //Inspection VBlock index
					IF (pInspVBlock.VBlock_Is_Occupied AND pInspVBlock.Inspection[idx_inspect_unit].Item_Inspection_Status = INSPECTION_RESULTS_NONESOFAR) THEN //Current vblock in front of inspection after index is occupied and hasn't been inspected yet
						//Handle resetting the VC object array datapoints to restart recording
//						brsmemset(ADR(pInspVCTrend.iInspectionGood[0]), 0, MAX_IDX_DISPENSE_VC_ARRAY + 1);
//						brsmemset(ADR(pInspVCTrend.iInspectionBad[0]), 0, MAX_IDX_DISPENSE_VC_ARRAY + 1);
//						brsmemset(ADR(pInspVCTrend.iInspectionError[0]), 0, MAX_IDX_DISPENSE_VC_ARRAY + 1);
//						brsmemset(ADR(pInspVCTrend.oInspectionTrigger[0]), 0, MAX_IDX_DISPENSE_VC_ARRAY + 1);
//						brsmemset(ADR(pInspVCTrend.oIlluminationTrigger[0]), 0, MAX_IDX_DISPENSE_VC_ARRAY + 1);
						InspVar.ii_VC_Trend_idx := 0;

						InspVar.Status := INSPECT_STATE_WAIT_VBLOCK_DISP;

					ELSIF pInspVBlock.VBlock_Is_Occupied AND pInspVBlock.Inspection[idx_inspect_unit].Item_Inspection_Status <> INSPECTION_RESULTS_NONESOFAR THEN
//						pInspVBlock.Error.Inspection_Error_1 := TRUE;
						Alarms.Inspection_Error_1 := TRUE;
//						pInspVBlock.Inspection[ii_inspect_units].Item_Inspection_Status := INSPECTION_ERROR_ALREADY_DONE;
						InspVar.Status := INSPECT_STATE_ERROR;
					END_IF;
				ELSIF InspVar.Flag_Inspect_Trigger_Now THEN //Force inspection to occur, i.e. manual trigger
//					//Handle resetting the VC object array datapoints to restart recording
//					brsmemset(ADR(pInspVCTrend.iInspectionGood[0]), 0, MAX_IDX_DISPENSE_VC_ARRAY + 1);
//					brsmemset(ADR(pInspVCTrend.iInspectionBad[0]), 0, MAX_IDX_DISPENSE_VC_ARRAY + 1);
//					brsmemset(ADR(pInspVCTrend.iInspectionError[0]), 0, MAX_IDX_DISPENSE_VC_ARRAY + 1);
//					brsmemset(ADR(pInspVCTrend.oInspectionTrigger[0]), 0, MAX_IDX_DISPENSE_VC_ARRAY + 1);
//					brsmemset(ADR(pInspVCTrend.oIlluminationTrigger[0]), 0, MAX_IDX_DISPENSE_VC_ARRAY + 1);
					InspVar.ii_VC_Trend_idx := 0;

					InspVar.Flag_Inspect_Trigger_Now := FALSE;

					bgTimerStart(InspVar.Timer.Timer_Inspection_Illum_DO_High, Tms(pInspCfg.Insp_Illum_ON_TO_S));
					bgTimerStart(InspVar.Timer.Timer_Inspection_Trigger_Wait, Tms(pInspCfg.Insp_Trigger_Wait_TO_S));

					InspVar.Status := INSPECT_STATE_WAIT_TRIG; //When triggering insp. manually, skip straight to waiting for the triggers rather than waiting for the vblock fractional displacement.
				ELSIF pInspectionIO.iInspectionBusy THEN //Shouldn't get a busy signal when not expecting it
					Alarms.Inspection_Busy_Without_Signal := TRUE;
					InspVar.Status := INSPECT_STATE_ERROR;
				ELSIF NOT pInspectionIO.iInspectionRunning THEN //Should always see DI corresponding to "running" state
					Alarms.Inspection_Not_Running := TRUE;
					InspVar.Status := INSPECT_STATE_ERROR;
				END_IF;
			ELSE//Inspection is disabled:
				InspVar.Status := INSPECT_STATE_DISABLED;
			END_IF;

		INSPECT_STATE_WAIT_VBLOCK_DISP:
			pInspectionIO.oInspectionTrigger := FALSE;
			pInspectionIO.oIlluminationTrigger := FALSE;

			IF InspVar.VBlock_Fract_Pos > pInspRec.Insp_VBlock_Displacement  THEN
				bgTimerStart(InspVar.Timer.Timer_Inspection_Illum_DO_High, Tms(pInspCfg.Insp_Illum_ON_TO_S));
				bgTimerStart(InspVar.Timer.Timer_Inspection_Trigger_Wait, Tms(pInspCfg.Insp_Trigger_Wait_TO_S));
				InspVar.Status := INSPECT_STATE_WAIT_TRIG;
			END_IF;

		INSPECT_STATE_WAIT_TRIG:
			pInspectionIO.oInspectionTrigger := FALSE;
			pInspectionIO.oIlluminationTrigger := NOT bgTimerIsTimeOut(InspVar.Timer.Timer_Inspection_Illum_DO_High);

			IF bgTimerIsTimeOut(InspVar.Timer.Timer_Inspection_Trigger_Wait) THEN
				bgTimerStart(InspVar.Timer.Timer_Inspection_Trigger_DO_High, Tms(pInspRec.Insp_Trigger_ON_TO_S));
				bgTimerStart(InspVar.Timer.Timer_Max_Insp_Busy_Signal, Tms(pInspCfg.Inspection_Max_Busy_TO_S));
				//
				InspVar.Status := INSPECT_STATE_WAIT_BUSY;
			ELSIF InspVar.VBlock_At_Inspect_Unit <> InspVar_LastCycle.VBlock_At_Inspect_Unit THEN
				Alarms.Inspection_VBlock_Idx_Waiting := TRUE;
				InspVar.Status := INSPECT_STATE_ERROR;
			END_IF;

		INSPECT_STATE_WAIT_BUSY:
			pInspectionIO.oInspectionTrigger := NOT bgTimerIsTimeOut(InspVar.Timer.Timer_Inspection_Trigger_DO_High);
			pInspectionIO.oIlluminationTrigger := NOT bgTimerIsTimeOut(InspVar.Timer.Timer_Inspection_Illum_DO_High);

			IF pInspectionIO.iInspectionBusy THEN
				bgTimerStart(InspVar.Timer.Timer_Inspection_Results_Wait, Tms(pInspCfg.Insp_Results_Wait_TO_S));
				InspVar.Status := INSPECT_STATE_WAIT_RESULTS;
			ELSIF bgTimerIsTimeOut(InspVar.Timer.Timer_Max_Insp_Busy_Signal) THEN
				Alarms.Insp_Err_Max_Busy_TO := TRUE;
				InspVar.Status := INSPECT_STATE_ERROR;
			ELSIF InspVar.VBlock_At_Inspect_Unit <> InspVar_LastCycle.VBlock_At_Inspect_Unit THEN
				Alarms.Inspection_VBlock_Idx_Waiting := TRUE;
				InspVar.Status := INSPECT_STATE_ERROR;
			END_IF;

		INSPECT_STATE_WAIT_RESULTS:
			pInspectionIO.oInspectionTrigger := NOT bgTimerIsTimeOut(InspVar.Timer.Timer_Inspection_Trigger_DO_High);
			pInspectionIO.oIlluminationTrigger := NOT bgTimerIsTimeOut(InspVar.Timer.Timer_Inspection_Illum_DO_High);

			IF NOT pInspectionIO.iInspectionBusy THEN
				pInspectionIO.oInspectionTrigger := FALSE;
				pInspectionIO.oIlluminationTrigger := FALSE;
				IF pInspectionIO.iInspectionError AND NOT pInspectionIO.iInspectionGood THEN
					pInspVBlock.Inspection[idx_inspect_unit].Item_Inspection_Status := INSPECTION_RESULTS_ERROR;
					pInspStats.Num_Err := pInspStats.Num_Err + 1;
				ELSE
					IF pInspectionIO.iInspectionGood THEN
						pInspVBlock.Inspection[idx_inspect_unit].Item_Inspection_Status := INSPECTION_RESULTS_GOOD;
						pInspStats.Num_Passed := pInspStats.Num_Passed + 1;

						pInspSeqFails := 0;
					ELSE
						pInspVBlock.Inspection[idx_inspect_unit].Item_Inspection_Status := INSPECTION_RESULTS_BAD;
						pInspStats.Num_Failed := pInspStats.Num_Failed + 1;

						pInspSeqFails := pInspSeqFails + 1;
					END_IF;
				END_IF;
				pInspVBlock.Inspection[idx_inspect_unit].Inspection_Time := bgTimerTimeElapsed(InspVar.Timer.Timer_Inspection_Results_Wait);
				//Return to state to wait for next inspection trigger event
				InspVar.Status := INSPECT_STATE_READY;
			ELSIF bgTimerIsTimeOut(InspVar.Timer.Timer_Inspection_Results_Wait) THEN
				//Failed to receive results within the specified timeout
				pInspectionIO.oInspectionTrigger := FALSE;
				pInspectionIO.oIlluminationTrigger := FALSE;

				pInspStats.Num_Unanswered := pInspStats.Num_Unanswered + 1;

				Alarms.Inspection_Results_TO_NoAnswer := TRUE;
				InspVar.Status := INSPECT_STATE_ERROR;
			ELSIF InspVar.VBlock_At_Inspect_Unit <> InspVar_LastCycle.VBlock_At_Inspect_Unit THEN
				Alarms.Inspection_VBlock_Idx_Waiting := TRUE;
				InspVar.Status := INSPECT_STATE_ERROR;
			END_IF;

		INSPECT_STATE_ERROR:

		INSPECT_STATE_DISABLED:
			IF pInspRec.Enable = 1 THEN
				InspVar.Status := INSPECT_STATE_INIT;
			END_IF;
	END_CASE;

	//Call timers
	bgTimerCyclic(InspVar.Timer.Timer_Inspection_Trigger_DO_High);
	bgTimerCyclic(InspVar.Timer.Timer_Inspection_Illum_DO_High);
	bgTimerCyclic(InspVar.Timer.Timer_Inspection_Results_Wait);
	bgTimerCyclic(InspVar.Timer.Timer_Inspection_Trigger_Wait);
	bgTimerCyclic(InspVar.Timer.Timer_Max_Insp_Busy_Signal);
//	bgTimerCyclic(InspectionRunSigBypass_ResetTime);

END_FUNCTION_BLOCK
```

### Library Logical/Application_Logic/pkgInspect/libInsp (IEC)

#### Insp_Enumerations.typ
```iecst
TYPE
	HERNON_Inspect_Enum :
		(
		INSPECT_STATE_INIT := 0,
		INSPECT_STATE_READY := 1,
		INSPECT_STATE_WAIT_RESULTS := 2,
		INSPECT_STATE_ERROR := 3,
		INSPECT_STATE_DISABLED := 4,
		INSPECT_STATE_WAIT_TRIG := 5,
		INSPECT_STATE_WAIT_BUSY := 6,
		INSPECT_STATE_WAIT_VBLOCK_DISP := 7,
		INSPECT_STATE_MANUAL := 8
		);
	HERNON_Inspect_Unit_ID_Enum :
		(
		INSPECT_PRIMER := 0,
		INSPECT_MOUTH := 1
		);
	HERNON_Inspection_Outcome_Enum :
		(
		INSPECTION_RESULTS_NONESOFAR := 0,
		INSPECTION_RESULTS_GOOD := 1,
		INSPECTION_RESULTS_BAD := 2,
		INSPECTION_RESULTS_ERROR := 3,
		INSPECTION_NA_EMPTY_VBLOCK := 4,
		INSPECTION_ERROR_ALREADY_DONE := 5
		);
END_TYPE
```

#### Insp_RecCfg.typ
```iecst
TYPE
	HERNON_Rec_Inspect_typ : 	STRUCT
		Enable : UDINT;
		Insp_Trigger_ON_TO_S : REAL;
		Insp_VBlock_Displacement : REAL;
		Sequential_Fails_Stop_Line : UDINT;
	END_STRUCT;
	HERNON_Cfg_Inspect_typ : 	STRUCT
		VBlock_Offset_From_PiP_Sensor : UDINT;
		Inspection_Max_Busy_TO_S : REAL;
		Insp_Results_Wait_TO_S : REAL;
		Insp_Trigger_Wait_TO_S : REAL;
		Insp_Illum_ON_TO_S : REAL;
	END_STRUCT;
END_TYPE
```

#### Insp_Alarms_Warnings.typ
```iecst
TYPE
	HERNON_Alarm_Inspect_typ : 	STRUCT
		Inspection_Error_1 : BOOL; (*0,1*)
		Inspection_Error_2 : BOOL; (*2,3*)
		Inspect_IO_Alloc_Error : BOOL; (*4,5*)
		Err_Insp_VBlock_Acc_Idx : BOOL; (*6,7*)
		Inspection_Not_Running : BOOL; (*8,9*)
		Inspection_Busy_Without_Signal : BOOL; (*10,11*)
		Insp_Err_Max_Busy_TO : BOOL; (*12,13*)
		Inspection_Results_TO_NoAnswer : BOOL; (*14,15*)
		Inspection_VBlock_Idx_Waiting : BOOL; (*16,17*)
		Inspect_Not_Ready_On_Start : BOOL; (*18*)
		Inspect_Error_During_Runtime : BOOL; (*19*)
		Inspection_Sequential_Fails : BOOL; (*20,21*)
	END_STRUCT;
END_TYPE
```

### Program Logical/Application_Logic/Control

#### Main.st
```iecst
PROGRAM _INIT

END_PROGRAM

PROGRAM _CYCLIC
	(* Insert code here *)

	CASE MachineState OF
		MACHINE_STATE_INIT:

		MACHINE_STATE_IDLE:

		MACHINE_STATE_RUNNING:

		MACHINE_STATE_ERRORSTOP:

		MACHINE_STATE_MANUAL_CTRL:

	END_CASE;

	CASE ProcessState OF
		PRCS_STATE_INIT:

		PRCS_STATE_IDLE:

		PRCS_STATE_WAIT_LOADER:

		PRCS_STATE_FEED_OFFSET:

		PRCS_STATE_BLADE_CREASER:

		PROCESS_STATE_FINISHING:

		PROCESS_STATE_ERROR:

	END_CASE;
END_PROGRAM

PROGRAM _EXIT
	(* Insert code here *)

END_PROGRAM
```

### Program Logical/Application_Logic/FeedRoller

#### Main.st
```iecst
PROGRAM _INIT
	(* Insert code here *)

END_PROGRAM

PROGRAM _CYCLIC

END_PROGRAM

PROGRAM _EXIT
	(* Insert code here *)

END_PROGRAM
```

### Package Logical/paiComponents - pai Components and Libraries

### bgdebug.h
```c
#ifndef _BG_DEBUG_H
#define _BG_DEBUG_H

#ifdef WIN32
#define DBG printf
#define DBGMSG printf

#define DBGCRT printf
#define DBGERR printf
#define DBGWAR printf
#define DBGINF printf
#define DBGDBG printf

#else

#include <bur/plc.h>
#include "bgringbuffer.h"

#define BG_DEBUG_LEVEL_CRITICAL		0
#define BG_DEBUG_LEVEL_ERROR		1
#define BG_DEBUG_LEVEL_WARNING		2
#define BG_DEBUG_LEVEL_INFO			3
#define BG_DEBUG_LEVEL_DEBUG		4

#define BG_DEBUG_UNUSED	0x0

/*
- To completly remove debug msgs from the source code use:
#define BG_DEBUG_ENABLE 0
*/
#define BG_DEBUG_ENABLE 1

/*ptr to global ring buffer for debug messages*/
_GLOBAL bgRingBuffer_typ gRingBuffer;

#if BG_DEBUG_ENABLE == 1
/*BG_DEBUG_ENABLE == 1 => debug messages present in the source code*/
#define DBG(format, args...)	bgRingBuffPutDbgInfo(&gRingBuffer, __FILE__, __FUNCTION__, BG_DEBUG_LEVEL_CRITICAL, BG_DEBUG_UNUSED, format, ## args);
#define DBGMSG(format, args...)	bgRingBuffPrintf(&gRingBuffer, format, ## args);

#define DBGCRT(format, args...)	bgRingBuffPutDbgInfo(&gRingBuffer, __FILE__, __FUNCTION__, BG_DEBUG_LEVEL_CRITICAL, BG_DEBUG_UNUSED, format, ## args);
#define DBGERR(format, args...)	bgRingBuffPutDbgInfo(&gRingBuffer, __FILE__, __FUNCTION__, BG_DEBUG_LEVEL_ERROR, BG_DEBUG_UNUSED, format, ## args);
#define DBGWAR(format, args...)	bgRingBuffPutDbgInfo(&gRingBuffer, __FILE__, __FUNCTION__, BG_DEBUG_LEVEL_WARNING, BG_DEBUG_UNUSED, format, ## args);
#define DBGINF(format, args...)	bgRingBuffPutDbgInfo(&gRingBuffer, __FILE__, __FUNCTION__, BG_DEBUG_LEVEL_INFO, BG_DEBUG_UNUSED, format, ## args);
#define DBGDBG(format, args...)	bgRingBuffPutDbgInfo(&gRingBuffer, __FILE__, __FUNCTION__, BG_DEBUG_LEVEL_DEBUG, BG_DEBUG_UNUSED, format, ## args);

#else
/*BG_DEBUG_ENABLE == 0 => all debug messages removed from the source code*/
#define DBG(format, args...)  ;
#define DBGMSG(format, args...)  ;

#define DBGCRT(format, args...)	;
#define DBGERR(format, args...)	;
#define DBGWAR(format, args...)	;
#define DBGINF(format, args...)	;
#define DBGDBG(format, args...)	;

#endif /*#if BG_DEBUG_ENABLE*/

#endif /*#ifdef WIN32*/

#endif /*#ifndef _BG_DEBUG_H*/
```

### bgPVSerializeJSON.c
```c
#ifndef _BG_SERIALIZEJSON_C
#define _BG_SERIALIZEJSON_C
/**
3/17/2015
-fixed serious bug that was causing incorrect setting of the integer PV types shorter than DINT/UDINT (i.e. SINT, USINT, INT, UINT)
*/
#ifdef WIN32
#include "string.h"
#else
#include <bur/plctypes.h>
#endif

//#include <string.h>
//#include <brsystem.h>
//#include <sys_lib.h>
//#include <asstring.h>
#include "bgstring.h"
#include "bgsprintf.h"
#include "bgsscanf.h"
#include "bgsscanf.c"

#define PV_SERIALIZEJSON_ITEM_DELIM_CRLF "\r\n"
#define PV_SERIALIZEJSON_ITEM_DELIM_COMMA ","
//#define PV_SERIALIZE_STR_MARKUP "'"
#define PV_SERIALIZEJSON_STR_MARKUP "'"

#define PV_SERIALIZEJSON_ERR_ZEROPTR -1
#define PV_SERIALIZEJSON_ERR_PVNOTFOUND -2
#define PV_SERIALIZEJSON_ERR_PVADRNOTFOUND -3
#define PV_SERIALIZEJSON_ERR_OBUFOVERFLOW -4

#define PV_SERIALIZEJSON_ERR_LAST -10

typedef struct bgPVSerializeJSON_typ
{
	char* toOutStream;
	UDINT lengthOutStream;
	DINT outputCharCount;
	DINT errorCode;
	DINT arrayIndexFrom;
	DINT arrayIndexTo;
	char* pItemDelim;
	char* pStrMarkup;
	DINT lastElement;

}bgPVSerializeJSON_typ;

static void bgPVSubStructSerializeJSON(bgPVSerializeJSON_typ* p, char* pvNameRoot, char* pvName, UINT dimension);
static void bgPVSerializeJSON(bgPVSerializeJSON_typ* p, char* pvNameRoot, char* pvName);
static void bgPVArraySerializeJSONRootToFrom(bgPVSerializeJSON_typ* p, char* pvNameRoot, int dimension, int isArrayOfStruct);

//#ifndef DBG
//#define DBG() ;
//#endif

#define PV_TYPE_MAX_INDEX	24
static const char *bgPVTypeStrings[PV_TYPE_MAX_INDEX + 1]={
	"STRUCT",	/*0*/
	"BOOL",		/*1*/
	"SINT",		/*2*/
	"INT",		/*3*/
	"DINT",		/*4*/
	"USINT",		/*5*/
	"UINT",		/*6*/
	"UDINT",		/*7*/
	"REAL",		/*8*/
	"STRING ",	/*9*/
	"ULINT",		/*10*/
	"DATETIME",	/*11*/
	"TIME",		/*12*/
	"DATE",		/*13*/
	"LREAL",		/*14*/
	"ARRAY",		/*15*/
	"TIME_OF_DAY",	/*16*/
	"BYTE",		/*17*/
	"WORD",		/*18*/
	"DWORD",	/*19*/
	"LWORD",	/*20*/
	"WSTRING",	/*21*/
	"?22",		/*22*/
	"LINT",		/*23*/
	};

static const char *bgGetPVTypeString(int pvTypeIndex){
	if(pvTypeIndex >= PV_TYPE_MAX_INDEX){
		return "TYPE=?";
	}

	return bgPVTypeStrings[pvTypeIndex];
}

static void bgGetPVValueText(char* pvValue, UDINT data_typ, UDINT data_len, UINT dimension, UDINT adr)
{
/*
	if( dimension != 1)
		DBG("TODO: display multidimensional values...");
*/
	switch(data_typ){
		case PB_DT_STRUCT:
			//DBG("TODO: display struct values...");
			break;
		case PB_DT_BOOL:
			bgsprintf(pvValue, "%d", *( (char*)adr ));
			break;
		case PB_DT_INT8:
			bgsprintf(pvValue, "%d", *( (char*)adr) );
			break;
		case PB_DT_INT16:
			bgsprintf(pvValue, "%d", *( (short*)adr ) );
			break;
		case PB_DT_INT32:
			bgsprintf(pvValue, "%d", *( (int*)adr ));
			break;
		case PB_DT_BYTE:
			bgsprintf(pvValue, "%u", *( (unsigned char*)adr));
			break;
		case PB_DT_WORD:
			bgsprintf(pvValue, "%u", *( (unsigned short*)adr));
			break;
		case PB_DT_LONG:
			bgsprintf(pvValue, "%u", *( (unsigned int*)adr));
			break;
		case PB_DT_FLOAT:
			{
				char temp[32];
				ftoa( *((float*)adr), (UDINT)temp);
				bgsprintf(pvValue, "%s", temp);
			}
			break;
		case PB_DT_VIS:
			bgsprintf(pvValue, "%s", (char*)adr );
			break;
		case PB_DT_OCTET:
			//DBG("TODO: display octet values...");
			break;
		case PB_DT_DATE:
			//DBG("TODO: display date values...");
			break;
		case PB_DT_TIME:
			//DBG("TODO: display time values...");
			break;
		case PB_DT_DIFF:
			//DBG("TODO: display time-diff values...");
			break;
		case 14://double
			{
				char temp[32];
				double value_double = *((double*)(adr));
				float value_float = (float)value_double;
				ftoa( value_float, (UDINT)temp);
				bgsprintf(pvValue, "%s", temp);
			}
			break;
		case PB_DT_ARRAY:
			//DBG("TODO: display array values...");
			break;
	}
}

static void bgSetPVValueText(char* pvValue, UDINT data_typ, UDINT data_len, UINT dimension, UDINT adr)
{
/*
	if( dimension != 1)
		DBG("TODO: display multidimensional values...");
*/
	switch(data_typ){
		case PB_DT_STRUCT:
			//DBG("TODO: set struct values...");
			break;
		case PB_DT_BOOL:
			*((char*)adr) = (char)atoi((UDINT)pvValue);
			break;
		case PB_DT_INT8:
			*((SINT*)adr) = (SINT)atoi((UDINT)pvValue);
			break;
		case PB_DT_INT16:
			*((INT*)adr) = (INT)atoi((UDINT)pvValue);
			break;
		case PB_DT_INT32:
			*((DINT*)adr) = (DINT)atoi((UDINT)pvValue);
			break;
		case PB_DT_BYTE:
			*((USINT*)adr) = (USINT)atoi((UDINT)pvValue);
			break;
		case PB_DT_WORD:
			*((UINT*)adr) = (UINT)atoi((UDINT)pvValue);
			break;
		case PB_DT_LONG:
			*((UDINT*)adr) = (UDINT)atoi((UDINT)pvValue);
			break;
		case PB_DT_FLOAT:
			{
				*((float*)adr) = atof((UDINT)pvValue);
			}
			break;
		case PB_DT_VIS:
			{
				int ii=0;
				//copy string
				//don't copy over the size of the dest buffer!
				//terminate properly
				char* src=(char*)pvValue;
				char* dst=(char*)adr;
				//DBG("GBTST= %s len=%d", src, data_len);
				for(ii=0; ii<data_len; ii++){
					dst[ii] = src[ii];
					//if end of src string > exit
					if(!src[ii])
						break;
				}
				//src longer than dst > terminate dst
				dst[data_len-1] = 0;
			}
			break;
		case PB_DT_OCTET:
			//DBG("TODO: display octet values...");
			break;
		case PB_DT_DATE:
			//DBG("TODO: display date values...");
			break;
		case PB_DT_TIME:
			//DBG("TODO: display time values...");
			break;
		case PB_DT_DIFF:
			//DBG("TODO: display time-diff values...");
			break;
		case 14://double
			{
				float value_float = atof((UDINT)pvValue);
				double value_double = (double)value_float;
				*((double*)adr) = value_double;
			}
			break;
		case PB_DT_ARRAY:
			//DBG("TODO: display array values...");
			break;
	}
}

int bgFindCharInStrRev(char *s, char chr)
{
	int ii;
	int lenStr;
	char *ptrStr;

	/*exit if null ptrs*/
	if(!s)
		return -1;

	lenStr = strlen(s);

	/*exit if zero strings*/
	if( !lenStr || !chr )
		return -1;

	/*search for char <chr> within the string <s> starting from the end*/
	for(ii=lenStr-1; ii>=0; ii--)
	{
		ptrStr = s + ii;
		if(*ptrStr == chr){
			return (ii);
		}
	}
	return -1;
}

static void bgPVWriteOutStream(bgPVSerializeJSON_typ* p, char* pvName, char* pvTextValue)
{
	int dotPosition;

	if(!p || !p->toOutStream || !pvTextValue || !p->pItemDelim)
		return;

	if(pvName){
		dotPosition = bgFindCharInStrRev(pvName, '.');
		if(dotPosition < 0){
			dotPosition=0; //dot not found > take the entire pvname
		}else{
			dotPosition += 1;//dot found > take only the pvname after the dot
		}

		brsstrcat((UDINT)p->toOutStream, (UDINT)PV_SERIALIZEJSON_STR_MARKUP);
		brsstrcat((UDINT)p->toOutStream, (UDINT)&pvName[dotPosition]);
		brsstrcat((UDINT)p->toOutStream, (UDINT)PV_SERIALIZEJSON_STR_MARKUP);
		brsstrcat((UDINT)p->toOutStream, (UDINT)"=");
		brsstrcat((UDINT)p->toOutStream, (UDINT)pvTextValue);

		p->outputCharCount += brsstrlen((UDINT)pvName);
		p->outputCharCount += 1; //  + '='
	}else{
		brsstrcat((UDINT)p->toOutStream, (UDINT)pvTextValue);
	}

	if(!p->lastElement){
		brsstrcat((UDINT)p->toOutStream, (UDINT)p->pItemDelim);	// delimiter "\r\n" or ","
	}
	p->outputCharCount += strlen(pvTextValue);
	if(!p->lastElement){
		p->outputCharCount += strlen(p->pItemDelim); //  + sizeof the delimiter string
	}

	if(p->outputCharCount >= (p->lengthOutStream - 100) ){//TODO: needs to be a better way to handle output buffer overflow
		p->errorCode = PV_SERIALIZEJSON_ERR_OBUFOVERFLOW;
		return;
	}
}

static bgTxtWriteOutStream(bgPVSerializeJSON_typ* p, char* pTxt)
{
	if(!p || !p->toOutStream || !pTxt)
		return;

	brsstrcat((UDINT)p->toOutStream, (UDINT)pTxt);

	p->outputCharCount += strlen(pTxt);

	if(p->outputCharCount >= (p->lengthOutStream - 100) ){//TODO: needs to be a better way to handle output buffer overflow
		p->errorCode = PV_SERIALIZEJSON_ERR_OBUFOVERFLOW;
		return;
	}
}

static int bgPVSerializeJSONIsArray(int data_typ, int data_len, int dimension)
{
	if(data_typ && (dimension > 1)){
		return 1;
	}
	return 0;
}

static void bgPVArraySerializeJSON(bgPVSerializeJSON_typ* p, char* pvNameRoot, char* pvName, int dimension, int isArrOfStruct)
{
	char pvArrNameRoot[128];
	bgPVSerializeJSON_typ pvSerObj;

	if(!pvName)
		return;

	bgTxtWriteOutStream(p, PV_SERIALIZEJSON_STR_MARKUP);
	bgTxtWriteOutStream(p, pvName);
	bgTxtWriteOutStream(p, PV_SERIALIZEJSON_STR_MARKUP);
	bgTxtWriteOutStream(p, "=");

	pvSerObj.toOutStream = p->toOutStream;
	pvSerObj.lengthOutStream = p->lengthOutStream;
	pvSerObj.outputCharCount = p->outputCharCount;
	pvSerObj.errorCode = 0;
	pvSerObj.arrayIndexFrom = 0;
	pvSerObj.arrayIndexTo = dimension - 1;
	pvSerObj.pItemDelim =  PV_SERIALIZEJSON_ITEM_DELIM_COMMA;
	pvSerObj.pStrMarkup =  PV_SERIALIZEJSON_STR_MARKUP;
	pvSerObj.lastElement = 0;

	brsstrcpy((UDINT)pvArrNameRoot, (UDINT)pvNameRoot);
	brsstrcat((UDINT)pvArrNameRoot, (UDINT)".");
	brsstrcat((UDINT)pvArrNameRoot, (UDINT)pvName);

	bgPVArraySerializeJSONRootToFrom(&pvSerObj, pvArrNameRoot, dimension, isArrOfStruct);

	p->outputCharCount = pvSerObj.outputCharCount;
	p->errorCode = pvSerObj.errorCode;

}

static void bgPVArraySerializeJSONRootToFrom(bgPVSerializeJSON_typ* p, char* pvNameRoot, int dimension, int isArrayOfStruct)
{
	int ii = 0;
	// TODO: checking for max size of the strings that are copied to these arrays
	char structName[256];
	char structItemName[32];
	DINT arrLastElement;
/*
Array of objects:
 "myarray" = "[
 {ID=0, HeadID=0, var={Type=0, Format=0}},
 {},
 {}]"

*/

	arrLastElement = p->lastElement;
	p->lastElement = 0;
	bgTxtWriteOutStream(p, "[");
	for(ii = p->arrayIndexFrom; (ii < dimension) && (ii <= p->arrayIndexTo); ii++){
		// NOTE: verify why PV_item destroys content of the buffer supplied as 1st param
		{
			char arrayIndexTxt[10];
			brsstrcpy((UDINT)structItemName, (UDINT)pvNameRoot);
			brsstrcat((UDINT)structItemName, (UDINT)"[");
			brsitoa(ii, (UDINT)arrayIndexTxt);
			brsstrcat((UDINT)structItemName, (UDINT)arrayIndexTxt);
			brsstrcat((UDINT)structItemName, (UDINT)"]");
		}

		if(isArrayOfStruct)
			bgTxtWriteOutStream(p, "{");

		if((ii == (dimension-1)) || (ii == p->arrayIndexTo) ){
			p->lastElement = 1;
		}

		bgPVSerializeJSON(p, structItemName, 0);

		if((ii == (dimension-1)) || (ii == p->arrayIndexTo) ){
			if(isArrayOfStruct)
				bgTxtWriteOutStream(p, "}");
		}else{
			if(isArrayOfStruct)
				bgTxtWriteOutStream(p, "},");
		}

		if(p->errorCode)
			return;
	}

	if(!isArrayOfStruct){
		//	p->outputCharCount -= strlen(p->pItemDelim);//workaroud: remove delim for the last array element
		//	p->toOutStream[p->outputCharCount] = 0;
	}

	bgTxtWriteOutStream(p, "]");
	p->lastElement = arrLastElement;

	if(!isArrayOfStruct && !p->lastElement){
		bgTxtWriteOutStream(p, p->pItemDelim);
	}

}

static void bgPVSerializeJSON(bgPVSerializeJSON_typ* p, char* pvNameRoot, char* pvName)
{
	UINT status;
	UDINT data_typ;
	UDINT data_len;
	UINT dimension;
	UDINT adr;
	char structItemPVName[256];

	if( !pvName){
		brsstrcpy((UDINT)structItemPVName, (UDINT)pvNameRoot);

	}else{
		brsstrcpy((UDINT)structItemPVName, (UDINT)pvNameRoot);
		brsstrcat((UDINT)structItemPVName, (UDINT)".");
		brsstrcat((UDINT)structItemPVName, (UDINT)pvName);
	}

	status = PV_ninfo(structItemPVName, &data_typ, &data_len, &dimension);

	if( status ){
		p->errorCode = status;
		return;
	}

	if( bgPVSerializeJSONIsArray(data_typ, data_len, dimension) ){
		bgPVArraySerializeJSON(p, pvNameRoot, pvName, dimension, (data_typ==PB_DT_ARRAY)?1:0);
		return;
	}

	status = PV_xgetadr(structItemPVName, &adr, &data_len);

	if( status ){
		p->errorCode = status;
		return;
	}

	if( (data_typ == PB_DT_STRUCT) ){
		//DBG("PV='%s' Typ=%s Len=%d Dim=%d" , pvnamecomplete, bgGetPVTypeString(data_typ), data_len, dimension);

		if( (dimension == 1) && (data_len==4)){
			//enum data type!!! > will be handled below as a UDINT
			data_typ = PB_DT_INT32;
		}else{
			bgPVSubStructSerializeJSON(p, pvNameRoot, pvName, dimension);
			return;
		}
	}

	{
		char pvTextValue[256];
		int len = 0;

		if(data_typ == PB_DT_VIS){//STRING VALUES ONLY > marked with a special markup at the begining and end
			brsstrcpy((UDINT)pvTextValue, (UDINT)p->pStrMarkup);//set string begining markup (i.e. "\"")
			len = strlen(pvTextValue);
		}

		bgGetPVValueText(&pvTextValue[len], data_typ, data_len, dimension, adr);

		if(data_typ == PB_DT_VIS){//STRING VALUES ONLY > marked with a special markup at the begining and end
			brsstrcat((UDINT)pvTextValue, (UDINT)p->pStrMarkup);//set string ending markup (i.e. "\"")
		}

		//DBG("stritemPV='%s' Typ=%s Len=%d Dim=%d Val=%s" , pvName, bgGetPVTypeString(data_typ), data_len, dimension, pvTextValue);
		bgPVWriteOutStream(p, pvName, pvTextValue);
	}

}

static void bgPVSubStructSerializeJSON(bgPVSerializeJSON_typ* p, char* pvNameRoot, char* pvName, UINT dimension)
{
/*
Example:
typedef struct str1_typ{
UINT val1;
UINT val2;
}str1_typ;

typedef struct str2_typ{
UINT val3;
}str2_typ;

typedef struct str3_typ{
UINT val4;
struct str1_typ s1;
struct str2_typ s2;
}str3_typ;

_GLOBAL str3_typ test;

All available PV Names are:
test.val4
test.s1.val1
test.s1.val2
test.s2.val3;

Top PV Name (pvNameRoot):
test

During iteration, followin values will appear for 'structItemName':
s1
s2
val4

During iteration, following values will appear for 'structItemPVNameNoRoot':
val4
s1.val1
s1.val2
s2.val3

*/
	int ii = 0;
	// TODO: checking for max size of the strings that are copied to these arrays
	char structName[256];
	char structItemName[32];
	char structItemPVNameNoRoot[256];
	UINT status;
	UDINT data_typ;
	UDINT data_len;
	UDINT adr;

	if(pvName){
		bgTxtWriteOutStream(p, PV_SERIALIZEJSON_STR_MARKUP);
		bgTxtWriteOutStream(p, pvName);
		bgTxtWriteOutStream(p, PV_SERIALIZEJSON_STR_MARKUP);
		bgTxtWriteOutStream(p, "={");
	}

	for(ii=0; ii < dimension; ii++){
		// NOTE: verify why PV_item destroys concent of the buffer supplied as 1st param
		if( !pvName){
			brsstrcpy((UDINT)structName, (UDINT)pvNameRoot);
		}else{
			brsstrcpy((UDINT)structName, (UDINT)pvNameRoot);
			brsstrcat((UDINT)structName, (UDINT)".");
			brsstrcat((UDINT)structName, (UDINT)pvName);
		}

		//DBG("1)bgPVSubStr.. ii=%d str=%s item=%s", ii, structName, structItemName);
		status = PV_item(structName, ii, structItemName);
		//DBG("2)bgPVSubStr.. ii=%d str=%s item=%s", ii, structName, structItemName);

		if(status && (status != 14713)){
			// TODO: error handling
			//DBG("bgPVSubStr.. ii=%d str=%s item=%s err=%d", ii, structName, structItemName, status);
			p->errorCode = status;
			return;
		}

		//DBG("item=%d, name=%s", ii, structItemName);
		// TODO: check for max length of the PV name
		if(!pvName){
			brsstrcpy((UDINT)structItemPVNameNoRoot, (UDINT)structItemName);
		}else{
			if(status == 14713){//14713 is to handle enum type??? find out if there is a better solutiuon
				//following code is to handle an enum type that is reported as a structure (type 0). However, there are no structure elements and is not clear how to access values???
				char pvTextValue[64];

				status = PV_ninfo(structName, &data_typ, &data_len, &dimension);
				status = PV_xgetadr(structName, &adr, &data_len);
				//based on the reported lenght, try to guess the type of the enum
				if(data_len == 1){
					data_typ = PB_DT_BYTE;
				}else
					if(data_len == 2){
					data_typ = PB_DT_WORD;
				}else{
					data_typ = PB_DT_LONG;
				}
				bgGetPVValueText(&pvTextValue[0], data_typ, data_len, dimension, adr);
				if(ii == (dimension - 1)){
					p->lastElement = 1;
				}
				else{
					p->lastElement = 0;
				}
				bgPVWriteOutStream(p, pvName, pvTextValue);
				return;
			}

			brsstrcpy((UDINT)structItemPVNameNoRoot, (UDINT)pvName);
			brsstrcat((UDINT)structItemPVNameNoRoot, (UDINT)".");
			brsstrcat((UDINT)structItemPVNameNoRoot, (UDINT)structItemName);
		}

		if(ii == (dimension - 1)){
			p->lastElement = 1;
		}
		else{
			p->lastElement = 0;
		}
		bgPVSerializeJSON(p, pvNameRoot, structItemPVNameNoRoot);

		if(p->errorCode)
			return;
	}

	if(pvName){
		bgTxtWriteOutStream(p, "}");
	}
}

DINT bgPVRootArraySerializeJSON(char* pvNameRoot, char* toOutStream, UDINT lengthOutStream, UDINT begIndex, UDINT endIndex)
{
	UINT status;
	UDINT data_typ;
	UDINT data_len;
	UINT dimension;
	UDINT adr;
	DINT outputCharCount = 0;

	bgPVSerializeJSON_typ pvSerObj;

	if(!pvNameRoot || !toOutStream){
		return PV_SERIALIZEJSON_ERR_ZEROPTR;
	}

	if(toOutStream){
		brsstrcpy((UDINT)toOutStream, (UDINT)"");
	}
	pvSerObj.toOutStream = toOutStream;
	pvSerObj.lengthOutStream = lengthOutStream;
	pvSerObj.outputCharCount = 0;
	pvSerObj.errorCode = 0;
	pvSerObj.arrayIndexFrom = begIndex;
	pvSerObj.arrayIndexTo = endIndex;
	pvSerObj.pItemDelim =  PV_SERIALIZEJSON_ITEM_DELIM_COMMA;
	pvSerObj.pStrMarkup =  PV_SERIALIZEJSON_STR_MARKUP;
	pvSerObj.lastElement = 0;

	status = PV_ninfo(pvNameRoot, &data_typ, &data_len, &dimension);
	if( status ){
		return PV_SERIALIZEJSON_ERR_PVNOTFOUND;
	}

	status = PV_xgetadr(pvNameRoot, &adr, &data_len);
	if( status ){
		return PV_SERIALIZEJSON_ERR_PVADRNOTFOUND;
	}

	if(data_typ == PB_DT_STRUCT){
		//DBG("TOPPV='%s' Typ=%s Len=%d Dim=%d" , pvNameRoot, bgGetPVTypeString(data_typ), data_len, dimension);
		bgPVSubStructSerializeJSON(&pvSerObj, pvNameRoot, 0, dimension);
	}else
	if(data_typ == PB_DT_ARRAY){
		bgPVArraySerializeJSONRootToFrom(&pvSerObj, pvNameRoot, dimension, 1, 0);
	}else
	if(data_typ == PB_DT_VIS){//visible string
		bgPVArraySerializeJSONRootToFrom(&pvSerObj, pvNameRoot, dimension, 0, 1);
	}else
	if( ((data_typ == PB_DT_INT16) || (data_typ == PB_DT_INT32) || (data_typ == PB_DT_WORD) || (data_typ == PB_DT_LONG))&& (dimension > 1)){//aray of INT16
		bgPVArraySerializeJSONRootToFrom(&pvSerObj, pvNameRoot, dimension, 0, 1);
	}else{
		char pvTextValue[64];
		bgGetPVValueText(&pvTextValue[0], data_typ, data_len, dimension, adr);
		//DBG("TOPPV NOT A STRUCT! PV='%s' Typ=%s Len=%d Dim=%d Val=%s" , pvNameRoot, bgGetPVTypeString(data_typ), data_len, dimension, pvTextValue);
	}

	if(pvSerObj.errorCode){
		if(pvSerObj.errorCode < 0){
			return pvSerObj.errorCode;
		}
		return (pvSerObj.errorCode * (-1));
	}

	return pvSerObj.outputCharCount;
}

DINT bgPVStructSerializeJSON(char* pvNameRoot, char* toOutStream, UDINT lengthOutStream)
{
	UINT status;
	UDINT data_typ;
	UDINT data_len;
	UINT dimension;
	UDINT adr;
	DINT outputCharCount = 0;
	bgPVSerializeJSON_typ pvSerObj;

	if(!pvNameRoot || !toOutStream){
		return PV_SERIALIZEJSON_ERR_ZEROPTR;
	}

	if(toOutStream){
		brsstrcpy((UDINT)toOutStream, (UDINT)"");
	}
	pvSerObj.toOutStream = toOutStream;
	pvSerObj.lengthOutStream = lengthOutStream;
	pvSerObj.outputCharCount = 0;
	pvSerObj.errorCode = 0;
	pvSerObj.pItemDelim =  PV_SERIALIZEJSON_ITEM_DELIM_CRLF;
	pvSerObj.pStrMarkup =  "";

	status = PV_ninfo(pvNameRoot, &data_typ, &data_len, &dimension);
	if( status ){
		return PV_SERIALIZEJSON_ERR_PVNOTFOUND;
	}

	status = PV_xgetadr(pvNameRoot, &adr, &data_len);
	if( status ){
		return PV_SERIALIZEJSON_ERR_PVADRNOTFOUND;
	}

	if(data_typ == PB_DT_STRUCT){
		//DBG("TOPPV='%s' Typ=%s Len=%d Dim=%d" , pvNameRoot, bgGetPVTypeString(data_typ), data_len, dimension);
		bgPVSubStructSerializeJSON(&pvSerObj, pvNameRoot, 0, dimension);
	}else
	if(data_typ == PB_DT_ARRAY){
		pvSerObj.arrayIndexFrom = 0;
		pvSerObj.arrayIndexTo = dimension - 1;
		bgPVArraySerializeJSONRootToFrom(&pvSerObj, pvNameRoot, dimension, 1, 0);
	}
	else{
		char pvTextValue[64];
		bgGetPVValueText(&pvTextValue[0], data_typ, data_len, dimension, adr);
		//DBG("TOPPV NOT A STRUCT! PV='%s' Typ=%s Len=%d Dim=%d Val=%s" , pvNameRoot, bgGetPVTypeString(data_typ), data_len, dimension, pvTextValue);
	}

	if(pvSerObj.errorCode){
		if(pvSerObj.errorCode < 0){
			return pvSerObj.errorCode;
		}
		return (pvSerObj.errorCode * (-1));
	}

	return pvSerObj.outputCharCount;
}

//Maximum number of PV-s per file that can be deserialized!!!
#define BGPV_DESER_MAXPVCOUNT 1000

DINT bgPVStructDeserializeJSON(char* pvNameRoot, char* fromStream, UDINT lengthStream)
{
	UDINT ii;
	bgStringListEx_typ lineList1;
	bgStringListEx_typ lineSplit1;
	char* memLineList[BGPV_DESER_MAXPVCOUNT];
	char* memLineSplit[10];
	char structItemPVName[256];

	UINT status;
	UDINT data_typ;
	UDINT data_len;
	UINT dimension;
	UDINT adr;
	UDINT errorCounter = 0;

	bgStringListLinesEx(&lineList1, fromStream, (char*)memLineList, BGPV_DESER_MAXPVCOUNT*sizeof(char*));
	for(ii=0; ii<lineList1.itemCount; ii++){
		//DBG("ln%d: %s", ii, lineList1.items[ii]);
		bgStringSplitLineEx(&lineSplit1, '=',  (char*)lineList1.items[ii], (char*)memLineSplit, (int)10*sizeof(char*));
		//DBG("ln%d: key=%s val=%s", ii, lineSplit1.items[0], lineSplit1.items[1]);

		brsstrcpy((UDINT)structItemPVName, (UDINT)pvNameRoot);
		brsstrcat((UDINT)structItemPVName, (UDINT)".");
		brsstrcat((UDINT)structItemPVName, (UDINT)lineSplit1.items[0]);

		//DBG("PV=%s Val=%s", structItemPVName, lineSplit1.items[1]);
		status = PV_ninfo(structItemPVName, &data_typ, &data_len, &dimension);

		if( status ){
			// TODO: error handling
			//DBG("bgPVStructDes. PV='%s'; Error#=%d", structItemPVName, status);
			errorCounter++;
			continue;
		}

		status = PV_xgetadr(structItemPVName, &adr, &data_len);

		if( status ){
			// TODO: error handling
			//DBG("bgPVStructDes. Address for PV='%s'; Error=%d", structItemPVName, status);
			errorCounter++;
			continue;
		}

		bgSetPVValueText((char*)lineSplit1.items[1], data_typ, data_len, dimension, adr);
	}

	// TODO: return value in case of errors; detected version changes, etc.

	return errorCounter;

}

#endif //_BG_SERIALIZE_C
/*EOF*/
```

- Library Logical/paiComponents/Libraries/bgringbuf (ANSIC) (no source held here)

### Program Logical/paiComponents/paiFileService/paiFS (ANSIC) - pai File Service (TK#8)

#### paiFile.h - pai FS configuration defines 
```c
/********************************************************************
 * COPYRIGHT -- HP
 ********************************************************************
 * File: paiFile.h
 * Author: goran
 * Created: March 19, 2014
 *******************************************************************/

#include <bur/plctypes.h>

/*
###############################################################################
PAI_CONFIGURATION_SECTION
Code below allows configuration for:
application file system
###############################################################################
*/

/*
###############################################################################
Defines, Consts
###############################################################################
*/
/*
NOTE: Using C: disk is not the best solution considering that system files are there.
However, using disk other then C: (i.e. D:, etc) for application stuff creates
issue with the ability to view/copy/access application files from windows (multiple partitions not supported, etc)

File structure used in this application is following:

Directory:
C://Data
is used for application specific stuff.
This directory holds following files:
machine configuration file - "appcfg.txt"
machine factory deafult configuration file - "appcfgfactory.txt");

a subdirectory (REC) of the above directory is used for storing recipes.
C://Data/Rec

*/

#define PAI_FS_DEVICE_ROOT		"CFDISK"

/*file device name*/
//#define FILE_DEVICE_NAME	"CFDISK"
//#define FILE_DEVICE_CONF	 "/DEVICE=F:\\"
//#define FILE_DEVICE_CONF	 "/DEVICE=C:\\"
/*#define FILE_DEVICE_CONF	 "/DEVICE=D:\\Temp"*/

//IMPORTANT:
//in order for the following conditional compilation to work properly, PLC object in the Configuration view
//must contain following defintion:
//Folder: Build
//Field: Additional Build Options
//Value: -D $(AS_CONFIGURATION)
//Using the above, name of the current AS configuration (i.e. PPC820_ARwin1) becomes
//a defined preprocessor name. As a result, it's possible to destinguish between different configurations!
#ifdef PPC820_ARwin1
//In case of ARwin target, disk access uses networking and the disk storage is on the windows side
//CRITICAL NOTE: following IP address must match the Windows IP address within the ARWin networking configuration
//#define FILE_DEVICE_CONF "/SIP=192.168.1.15 /PROTOCOL=cifs /SHARE=abc /USER=abc /PASSWORD=abc"
#define FILE_DEVICE_CONF "/SIP=192.168.100.2 /PROTOCOL=cifs /SHARE=E_Data /USER=gainco /PASSWORD=gainco"
#warning "paiFS - ARwin target!"
#endif

#ifdef PPC820_ARwin
//In case of ARwin target, disk access uses networking and the disk storage is on the windows side
//CRITICAL NOTE: following IP address must match the Windows IP address within the ARWin networking configuration
//#define FILE_DEVICE_CONF "/SIP=192.168.1.15 /PROTOCOL=cifs /SHARE=abc /USER=abc /PASSWORD=abc"
#define FILE_DEVICE_CONF "/SIP=192.168.100.2 /PROTOCOL=cifs /SHARE=E_Data /USER=gainco /PASSWORD=gainco"
#warning "paiFS - ARwin target!"
#endif

//#ifndef FILE_DEVICE_CONF
#ifndef PAI_FS_DEVICE_ROOT_CFG
//For all other target (i.e ARsim and ARemb), storage resides on a physical disk present in the system
//#define FILE_DEVICE_CONF	 "/DEVICE=C:\\"
#define PAI_FS_DEVICE_ROOT_CFG	"/DEVICE=C:\\"
#warning "paiFS - NONE ARwin target!"
#warning "Please verify File System configuration in paiFS.h"
#endif

//===================================================================================
//Define application directories
//Dirs are located at PAI_FS_DEVICE_ROOT
#define PAI_FS_APP_DIR_DATA		"Data"
#define PAI_FS_APP_DIR_CFG		"Data/Cfg"
#define PAI_FS_APP_DIR_REC		"Data/Rec"

//===================================================================================
//Define application devices
//Devices are dedicated dirs at PAI_FS_DEVICE_ROOT to be used for specific purpose
#define PAI_FS_DEVICE_CFG	"CONFIG"
#define PAI_FS_DEVICE_CFG_CFG "/DEVICE=C:/Data/Cfg"

#define PAI_FS_DEVICE_REC	"RECIPES"
#define PAI_FS_DEVICE_REC_CFG "/DEVICE=C:/Data/Rec"

#define PAI_FS_DEVICE_REC_PALLETE	"FILESPALLETE"
#define PAI_FS_DEVICE_REC_PALLETE_CFG "/DEVICE=C:/Data/Rec/Pallets"

#define PAI_FS_DEVICE_REC_LAYER	"FILESLAYERS"
#define PAI_FS_DEVICE_REC_LAYER_CFG "/DEVICE=C:/Data/Rec/Layers"

#define PAI_FS_DEVICE_USB	"USB"
#define PAI_FS_DEVICE_USB_CFG "/DEVICE=C:/Data/Rec"
```

- Program Logical/paiComponents/paiFileService/paiFSUnitTest (ANSIC) - Example application code for using PAI file service. (no source held here)

### paiPVSerDesMgr.c - pai SerDes Manager
```c
/********************************************************************
 * COPYRIGHT --
 ********************************************************************
 * Package: paiFileService
 * File: paiPVSerDesMgr.c
 * Author: goran
 * Created: August 18, 2015
 *******************************************************************/

#include <bur/plctypes.h>
#ifdef _DEFAULT_INCLUDES
	#include <AsDefault.h>
#endif

#include "../bglib/bgPVSerialize.h"
#include "paiPVSerDesMgr.h"
#include "paiFSInterface.h"
/*
###############################################################################
Functions
###############################################################################
*/
/**
captureCurrentTimeStamp()
-captures current datetime, converts it to a string a places the result string into a user supplied
text buffer (pDst, dstSize)
*/
static void captureCurrentTimeStamp(char* pDst, UDINT dstSize)
{

	char txt_yyyy[8];
	char txt_mo[8];
	char txt_dd[8];
	char txt_hh[8];
	char txt_mm[8];
	char txt_ss[8];
	char txt_ms[8];

	if(!pDst)
		return;

	DTStructureGetTime_typ DTStrGetTime_1;
	DTStructure DTStruc;

	DTStrGetTime_1.enable = 1;
	DTStrGetTime_1.pDTStructure = (UDINT)&DTStruc;
	DTStructureGetTime(&DTStrGetTime_1);

	brsitoa(DTStruc.year, (UDINT)txt_yyyy);
	brsitoa(DTStruc.month, (UDINT)txt_mo);
	brsitoa(DTStruc.day, (UDINT)txt_dd);
	brsitoa(DTStruc.hour, (UDINT)txt_hh);
	brsitoa(DTStruc.minute, (UDINT)txt_mm);
	brsitoa(DTStruc.second, (UDINT)txt_ss);
	brsitoa(DTStruc.millisec, (UDINT)txt_ms);

	//sprintf(pDst, "%02d %02d %04d %02d:%02d:%02d", DTStruc.month, DTStruc.day, DTStruc.year, DTStruc.hour, DTStruc.minute, DTStruc.second);
	brsstrcpy((UDINT)pDst, (UDINT)txt_yyyy);
	brsstrcat((UDINT)pDst, (UDINT)"-");
	brsstrcat((UDINT)pDst, (UDINT)txt_mo);
	brsstrcat((UDINT)pDst, (UDINT)"-");
	brsstrcat((UDINT)pDst, (UDINT)txt_dd);
	brsstrcat((UDINT)pDst, (UDINT)" ");
	brsstrcat((UDINT)pDst, (UDINT)txt_hh);
	brsstrcat((UDINT)pDst, (UDINT)":");
	brsstrcat((UDINT)pDst, (UDINT)txt_mm);
	brsstrcat((UDINT)pDst, (UDINT)":");
	brsstrcat((UDINT)pDst, (UDINT)txt_ss);
	brsstrcat((UDINT)pDst, (UDINT)".");
	brsstrcat((UDINT)pDst, (UDINT)txt_ms);
}
/*
###############################################################################
PV Serialize / Deserialize Mgr
###############################################################################
*/

static void paiPVInitAtPowerUpCyclicSetStatus(char* pStatus, char* pText)
{
	brsstrcpy((UDINT)pStatus, (UDINT)pText);
}

static void paiPVInitAtPowerUpCyclic(paiPVSerDesMgr_typ* p)
{
	int ii;

	if(!p)
		return;

	for(ii=0; ii < p->iItemCount; ii++){
		if(p->pvItems[ii].optInitAtPowerUp.oInitReady)
			continue;

		//0-nothing to do
		if(p->pvItems[ii].optInitAtPowerUp.iPowerUpConfig == 0){
			p->pvItems[ii].optInitAtPowerUp.oInitReady = 1;
			paiPVInitAtPowerUpCyclicSetStatus(p->pvItems[ii].optInitAtPowerUp.oStatus, "off");
			continue;
		}

		//1-use test data, if diff, execute just default function
		if(p->pvItems[ii].optInitAtPowerUp.iPowerUpConfig == 1){
			//check test data validity
			if(!p->pvItems[ii].optInitAtPowerUp.pTestDataStorage ||
				!p->pvItems[ii].optInitAtPowerUp.iTestData){
				p->pvItems[ii].optInitAtPowerUp.oError = 1;
				continue;
			}

			//check if callback function defined
			if(!p->pvItems[ii].pCallbackDefault){
				p->pvItems[ii].optInitAtPowerUp.oError = 2;
				continue;
			}

			//compare test data
			if( (*(UDINT*)(p->pvItems[ii].optInitAtPowerUp.pTestDataStorage)) != p->pvItems[ii].optInitAtPowerUp.iTestData ){
				//difference!!! > execute default function
				void (*fDefault)() =  ( void(*) () ) p->pvItems[ii].pCallbackDefault;
				(*fDefault)();
				p->pvItems[ii].optInitAtPowerUp.oInitReady = 1;
				paiPVInitAtPowerUpCyclicSetStatus(p->pvItems[ii].optInitAtPowerUp.oStatus, "test+dflt");
			}else{
				p->pvItems[ii].optInitAtPowerUp.oInitReady = 1;
				paiPVInitAtPowerUpCyclicSetStatus(p->pvItems[ii].optInitAtPowerUp.oStatus, "test+n.a.");
			}

			//write test data to data storage
			*((UDINT*)p->pvItems[ii].optInitAtPowerUp.pTestDataStorage) = p->pvItems[ii].optInitAtPowerUp.iTestData;
			continue;
		}

		//2-use test data, if diff, execute default function then restore data from file
		if(p->pvItems[ii].optInitAtPowerUp.iPowerUpConfig == 2){
			//check test data validity
			if(!p->pvItems[ii].optInitAtPowerUp.pTestDataStorage ||
			!p->pvItems[ii].optInitAtPowerUp.iTestData){
				p->pvItems[ii].optInitAtPowerUp.oError = 1;
				continue;
			}

			//check if callback function defined
			if(!p->pvItems[ii].pCallbackDefault){
				p->pvItems[ii].optInitAtPowerUp.oError = 2;
				continue;
			}

			//compare test data
			if( *((UDINT*)p->pvItems[ii].optInitAtPowerUp.pTestDataStorage) != p->pvItems[ii].optInitAtPowerUp.iTestData ){
				//difference!!! > execute default function
				void (*fDefault)() =  ( void(*) () ) p->pvItems[ii].pCallbackDefault;
				(*fDefault)();
				//p->pvItems[ii].optInitAtPowerUp.oInitReady = 1;
				paiPVInitAtPowerUpCyclicSetStatus(p->pvItems[ii].optInitAtPowerUp.oStatus, "test+dflt");
				//now, request read from file
				p->pvItems[ii].iDesRequest = 1;
			}else{
				paiPVInitAtPowerUpCyclicSetStatus(p->pvItems[ii].optInitAtPowerUp.oStatus, "test+n.a.");
				p->pvItems[ii].optInitAtPowerUp.oInitReady = 1;
			}

			//write test data to data storage
			*((UDINT*)p->pvItems[ii].optInitAtPowerUp.pTestDataStorage) = p->pvItems[ii].optInitAtPowerUp.iTestData;
			continue;
		}
	}
}

static void paiPVChangeMonitorInit(paiPVSerDesMgr_typ* p)
{

}

static void paiPVChangeMonitorCyclic(paiPVSerDesMgr_typ* p)
{
int ii;

	if(!p)
		return;

	for(ii=0; ii < p->iItemCount; ii++){

		//HMI DesRequest (i.e. Read PV from file request via HMI)
		if(!p->pvItems[ii].iDesRequest && (p->pvItems[ii].optPtrHMIData && p->pvItems[ii].optPtrHMIData->iBtnDesRequest)){
			p->pvItems[ii].optPtrHMIData->iBtnDesRequest = 0;
			p->pvItems[ii].iDesRequest = 1;
			continue;
		}

		//HMI SerRequest (i.e. Write PV to file request via HMI)
		if(!p->pvItems[ii].iSerRequest && (p->pvItems[ii].optPtrHMIData && p->pvItems[ii].optPtrHMIData->iBtnSerRequest)){
			p->pvItems[ii].optPtrHMIData->iBtnSerRequest = 0;
			p->pvItems[ii].iSerRequest = 1;
			continue;
		}

		//check if feature PV change monitoring feature is enabled for an item
		if(!p->pvItems[ii].optChangeMonitor.iChngEnable)
			continue;

		if(!p->pvItems[ii].pPV || !p->pvItems[ii].iPVSize){
			p->pvItems[ii].optChangeMonitor.oError = 3;
			continue;
		}

		if(!p->pvItems[ii].optChangeMonitor.pChangeMonitorMem){
			p->pvItems[ii].optChangeMonitor.oError = 1;
			continue;
		}

		if(p->pvItems[ii].iPVSize > p->pvItems[ii].optChangeMonitor.iChangeMonitorMemSize ){
			p->pvItems[ii].optChangeMonitor.oError = 2;
			continue;
		}

		if(p->pvItems[ii].optChangeMonitor.oState == 0){
			//init state > copy PV to private memory, begin change monitor
			brsmemcpy((UDINT)p->pvItems[ii].optChangeMonitor.pChangeMonitorMem, (UDINT)p->pvItems[ii].pPV, p->pvItems[ii].iPVSize);

			p->pvItems[ii].optChangeMonitor.iChngAccepted = 0;
			p->pvItems[ii].optChangeMonitor.iChngRejected = 0;
			p->pvItems[ii].optChangeMonitor.oChngDetected = 0;

			p->pvItems[ii].optChangeMonitor.oState = 1;
		}

		if(p->pvItems[ii].optChangeMonitor.oState == 1){

			//working state > monitor PV changes
			if( !brsmemcmp((UDINT)p->pvItems[ii].optChangeMonitor.pChangeMonitorMem, (UDINT)p->pvItems[ii].pPV, p->pvItems[ii].iPVSize) ){
				p->pvItems[ii].optChangeMonitor.oChngDetected = 0;
				if(p->pvItems[ii].optPtrHMIData){
					//HMI is defined
					p->pvItems[ii].optPtrHMIData->oBtnVisible = 1;//not visible
				}
				continue;
			}
			//change detected!
			p->pvItems[ii].optChangeMonitor.oChngDetected = 1;
			if(p->pvItems[ii].optPtrHMIData){
				//HMI is defined
				p->pvItems[ii].optPtrHMIData->oBtnVisible = p->pvItems[ii].optChangeMonitor.oChngDetected ? 0 : 1;
			}

			if(p->pvItems[ii].optChangeMonitor.iChngRejected || (p->pvItems[ii].optPtrHMIData && p->pvItems[ii].optPtrHMIData->iBtnChangeReject)){
				p->pvItems[ii].optChangeMonitor.iChngRejected = 0;
				if(p->pvItems[ii].optPtrHMIData){
					//HMI is defined
					p->pvItems[ii].optPtrHMIData->iBtnChangeReject = 0;
				}

				//restore changes from the private memory
				memcpy(p->pvItems[ii].pPV, p->pvItems[ii].optChangeMonitor.pChangeMonitorMem, p->pvItems[ii].iPVSize);
			}

			if(!p->pvItems[ii].iSerRequest && (p->pvItems[ii].optChangeMonitor.iChngAccepted ||
				(p->pvItems[ii].optPtrHMIData && p->pvItems[ii].optPtrHMIData->iBtnChangeAccept))){
				p->pvItems[ii].optChangeMonitor.iChngAccepted = 0;
				if(p->pvItems[ii].optPtrHMIData){
					//HMI is defined
					p->pvItems[ii].optPtrHMIData->iBtnChangeAccept = 0;
				}
				p->pvItems[ii].iSerRequest = 1;
				//update private memory
				memcpy(p->pvItems[ii].optChangeMonitor.pChangeMonitorMem, p->pvItems[ii].pPV, p->pvItems[ii].iPVSize);
			}
		}
	}
}

/*
Callback routine for paiPVSerDesMgr manager used for processing paiPVSerDesDesFromFile request.
This routine will be invoked following a file RD request.
The file data is deserialized into a provided PV within this function.
IMPORTANT:
- to handle a posibility for either file read error or deserialize error, make sure that the
given PV variable is initialized to default values before this request is executed.
*/
void paiCBReadFileDesPV(paiFileService_typ* p, UDINT pCallbackData)
{
DINT errCount;
paiPVSerDesMgr_typ* pPVSerDesMgr;
int ii;

	if(!p || !pCallbackData){
//		DBG(lgr,"cbReadFileDesPV: err: pCallbackData=0!");
		return;
	}

	pPVSerDesMgr = (paiPVSerDesMgr_typ*)pCallbackData;
	ii = pPVSerDesMgr->oState;

	captureCurrentTimeStamp(&pPVSerDesMgr->pvItems[ii].oTimestampLastDes[0], sizeof(pPVSerDesMgr->pvItems[ii].oTimestampLastDes));

	//read error?
	if(p->o.status){
		pPVSerDesMgr->pvItems[ii].oDesCount++;
		pPVSerDesMgr->pvItems[ii].oErrorCount++;
		pPVSerDesMgr->pvItems[ii].oError = p->o.status;
		//read error for a config file > file does not exist > use defaults!
		//gConfigApp.out.readcountererr++;
//		DBG(lgr,"cbReadFileDesPV: fileRD err (%s, %d)", pPVSerDesMgr->pvItems[ii].iFilename, p->o.status);

		//DBG(lgr,"cfg RD error=%d", paiFS.o.status);
//		DBG(lgr,"cbReadFileDesPV: Using cfg defaults");
		// TODO: nofify machine operator
		return;
	}

//	DBG(lgr,"cbReadFileDesPV: fileRD OK (%s)", pPVSerDesMgr->pvItems[ii].iFilename);

	pPVSerDesMgr->pvItems[ii].oDesCount++;
	pPVSerDesMgr->pvItems[ii].oFilesizeLastDes = p->o.bytecount;

	errCount = bgPVStructDeserialize(pPVSerDesMgr->pvItems[ii].iPVName, (char*)pPVSerDesMgr->pvItems[ii].pFilebuffer, p->prv.file.readex.bytesread);
	if(errCount){
//		DBG(lgr,"cbReadFileDesPV: des err(%d); struct change?", errCount);
	}

	//write test data to data storage if this option is enabled/defined
	if(!pPVSerDesMgr->pvItems[ii].optInitAtPowerUp.oInitReady && pPVSerDesMgr->pvItems[ii].optInitAtPowerUp.pTestDataStorage && pPVSerDesMgr->pvItems[ii].optInitAtPowerUp.iTestData){
		*((UDINT*)pPVSerDesMgr->pvItems[ii].optInitAtPowerUp.pTestDataStorage) = pPVSerDesMgr->pvItems[ii].optInitAtPowerUp.iTestData;
		paiPVInitAtPowerUpCyclicSetStatus(pPVSerDesMgr->pvItems[ii].optInitAtPowerUp.oStatus, "test+dflt+fRD");
		pPVSerDesMgr->pvItems[ii].optInitAtPowerUp.oInitReady = 1;
	}

	//Reset change monitor
	pPVSerDesMgr->pvItems[ii].optChangeMonitor.oState = 0;

}

void paiCBWriteFileSerPV(paiFileService_typ* p, UDINT pCallbackData)
{
paiPVSerDesMgr_typ* pPVSerDesMgr;
int ii;

	if(!p || !pCallbackData){
//		DBG(lgr,"cbWriteFileSerPV: err: pCallbackData=0!");
		return;
	}

	pPVSerDesMgr = (paiPVSerDesMgr_typ*)pCallbackData;
	ii = pPVSerDesMgr->oState;

	captureCurrentTimeStamp(&pPVSerDesMgr->pvItems[ii].oTimestampLastSer[0], sizeof(pPVSerDesMgr->pvItems[ii].oTimestampLastSer));

	//write error?
	if(p->o.status){
		pPVSerDesMgr->pvItems[ii].oErrorCount++;
		pPVSerDesMgr->pvItems[ii].oError = p->o.status;
		//read error for a config file > file does not exist > use defaults!
		//gConfigApp.out.readcountererr++;
//		DBG(lgr,"cbWriteFileSerPV: fileRD err (%s, %d)", pPVSerDesMgr->pvItems[ii].iFilename, p->o.status);

		//DBG(lgr,"cfg RD error=%d", paiFS.o.status);
//		DBG(lgr,"cbWriteFileSerPV: Using cfg defaults");
		// TODO: nofify machine operator
		return;
	}

//	DBG(lgr,"cbWriteFileSerPV: fileRD OK (%s)", pPVSerDesMgr->pvItems[ii].iFilename);
}

static BOOL paiPVSerDesSerToFile(paiPVSerDesMgr_typ* p, char* pvName, char* fileDeviceName, char* fileName, UDINT pBuffer, UDINT bufSize, UDINT pCallbackSer)
{
	DINT jj;
	DINT charsWritten;

	if(!p || !pvName || !fileName || !pBuffer || !bufSize)
		return 0;

	jj = p->oState;
	charsWritten = bgPVStructSerialize(pvName, (char*)pBuffer, bufSize);
	if(  charsWritten > 0){
//		DBG(lgr,"WRrec %s size=%d", fileName, charsWritten);
		p->pvItems[jj].oFilesizeLastSer = charsWritten;
		p->pvItems[jj].oSerCount++;
		paiFSFileWrRequest((paiFileService_typ*) p->pPaiFS, (UDINT) fileDeviceName, (UDINT)fileName, (UDINT)pBuffer, charsWritten, (UDINT) pCallbackSer, (UDINT) p);
		return 1;
	}else{
		p->pvItems[jj].oSerCount++;
		p->pvItems[jj].oErrorCount++;
//		DBG(lgr,"Can't serialize pv=%s", pvName);
		return 0;
	}
}

static void paiPVSerDesDesFromFile(paiPVSerDesMgr_typ* p, char* pvName, char* fileDeviceName, char* fileName, UDINT pBuffer, UDINT bufSize, UDINT pCallbackDes)
{
	paiFSFileRdRequest((paiFileService_typ*)p->pPaiFS, (UDINT) fileDeviceName, (UDINT)fileName, (UDINT)pBuffer, bufSize, (UDINT) pCallbackDes, (UDINT) p);
}

static BOOL paiPVSerDesIsItemDataOk(paiPVSerDesMgr_typ* p, int jj)
{
	//jj - current item index
	if(	!p->pvItems[jj].iPVName[0] ||
		!p->pvItems[jj].pPV ||
		!p->pvItems[jj].iPVSize ||
		!p->pvItems[jj].iFilename[0] ||
		!p->pvItems[jj].iDevicename[0] ||
		!p->pvItems[jj].pFilebuffer ||
		!p->pvItems[jj].iFilebufferSize){
		return 0; //not ok
	}

	return 1; //ok
}

void paiPVSerDesMgrInit(paiPVSerDesMgr_typ* p)
{
	if(!p || !p->iItemCount || (p->iItemCount > (PAI_FS_SERDESMGR_MAXITEMIDX+1)))
		return;

	//PV Change Monitor - init
	paiPVChangeMonitorInit(p);
}

void paiPVSerDesMgrCyclic(paiPVSerDesMgr_typ* p)
{
int ii;
int jj;

	//check params
	if(!p || !p->pPaiFS || !p->iItemCount || (p->iItemCount > (PAI_FS_SERDESMGR_MAXITEMIDX+1)))
		return;

	//PV InitAtPowerUp option
	paiPVInitAtPowerUpCyclic(p);

	//PV Change Monitor - cyclic
	paiPVChangeMonitorCyclic(p);

	//nothing to do if paiFS is busy
	if( paiFSFileRequestIsBusy((paiFileService_typ*)p->pPaiFS) )
		return;

	//check current item beeing processed
	if(p->oState >= p->iItemCount ){
		p->oState = 0;
	}

	//scan for serialize / deserialize requests
	for(ii = 0, jj = p->oState; ii < p->iItemCount; ii++){

		if(p->pvItems[jj].iSerRequest){
			p->pvItems[jj].iSerRequest = 0;
			if( paiPVSerDesIsItemDataOk(p, jj) ){
				p->oState = jj;
				paiPVSerDesSerToFile(p, (char*)p->pvItems[jj].iPVName,(char*)p->pvItems[jj].iDevicename, (char*)p->pvItems[jj].iFilename, (UDINT)p->pvItems[jj].pFilebuffer, p->pvItems[jj].iFilebufferSize, (UDINT) p->pvItems[jj].pCallbackSer);
				break;
			}else{
				p->pvItems[jj].oError = 1;
				brsstrcpy((UDINT)p->pvItems[jj].oErrorTxt, (UDINT)"paiPVSerDesSerToFile: Invalid Input Params" );
			}
		}

		if(p->pvItems[jj].iDesRequest){
			p->pvItems[jj].iDesRequest = 0;
			if( paiPVSerDesIsItemDataOk(p, jj) ){
				p->oState = jj;
				paiPVSerDesDesFromFile(p, (char*)p->pvItems[jj].iPVName,(char*)p->pvItems[jj].iDevicename, (char*)p->pvItems[jj].iFilename, (UDINT)p->pvItems[jj].pFilebuffer, p->pvItems[jj].iFilebufferSize, (UDINT) p->pvItems[jj].pCallbackDes);
				break;
			}else{
				p->pvItems[jj].oError = 1;
				brsstrcpy((UDINT)p->pvItems[jj].oErrorTxt, (UDINT)"paiPVSerDesDesFromFile: Invalid Input Params" );
			}
		}

		if(++jj >= p->iItemCount){
			jj = 0;
		}
	}
}
//eof
```

### Constants.var
```iecst
VAR CONSTANT
	paiHMI_ENUM_MENU_ITEMS_LT : DINT := 14;
	paiHMI_ENUM_TABS_MAXIDX : DINT := 14;
	paiHMI_ENUM_TG_TEXT_MAXIDX : DINT := 127;
	paiHMI_ENUM_TG_TEXT_MAXLEN : DINT := 31;
	paiHMI_PWD_LEVELS : DINT := 5;
	paiHMI_PWD_MAXLEN : DINT := 15;
END_VAR
(*Insert your comment here.*)
VAR CONSTANT
	paiHMI_ENUM_RUNMSG_MAXLEN : DINT := 255;
END_VAR
(*Insert your comment here.*)
VAR CONSTANT
	paiHMI_ENUM_MENU_ITEMS_RT : DINT := 10;
END_VAR
```
